KUKA KRL program: MyProgram_276().src

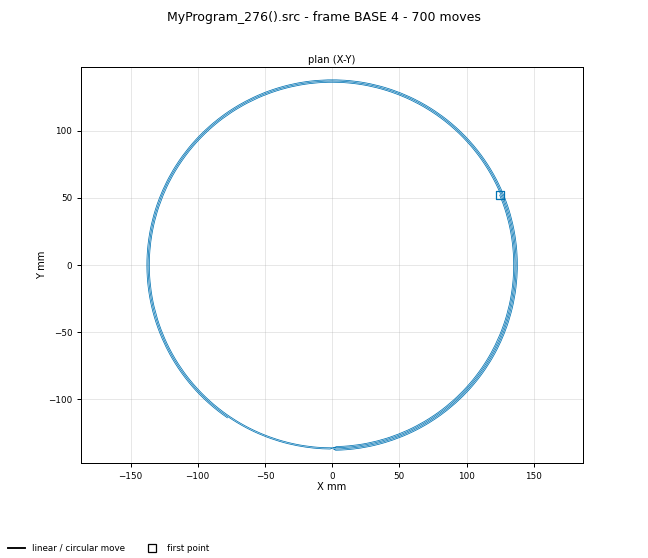
[picture p0: tool path of MyProgram_276().src in frame BASE 4, 700 of 700 moves have a stored position in this frame; points joined in program order, loops and branches not executed]
&ACCESS RVP
&REL 1
&PARAM TEMPLATE = C:\KRC\Roboter\Template\vorgabe
&PARAM EDITMASK = *
DEF MyProgram_276()
; ---- Setting reference (Base) ----
$BASE = BASE_DATA[4]

; --------------------------
; ---- Setting tool (TCP) ----
$TOOL = TOOL_DATA[3]
; --------------------------

$VEL.CP = VEL_APROX_PRINT
Startdeposition()
$VEL.CP = VEL_PRINT
LIN {X 124.6585,Y 52.0418,Z 172,A 23.3932,B 9.0147,C 0.1678,E1 9.1642,E2 428.0364} C_DIS
LIN {X 126.9033,Y 46.3017,Z 172,A 20.6618,B 9.0145,C 0.1775,E1 9.167,E2 430.7839} C_DIS
LIN {X 128.4598,Y 41.7937,Z 172,A 18.3883,B 9.0143,C 0.1885,E1 9.169,E2 433.0895} C_DIS
LIN {X 129.5892,Y 38.1419,Z 172,A 17.2072,B 9.0143,C 0.1833,E1 9.1699,E2 434.2181} C_DIS
LIN {X 130.4857,Y 34.952,Z 172,A 15.8377,B 9.0143,C 0.1864,E1 9.1709,E2 435.5844} C_DIS
LIN {X 131.283,Y 31.8269,Z 172,A 14.4299,B 9.0143,C 0.1911,E1 9.1719,E2 436.9981} C_DIS
LIN {X 132.2099,Y 27.7366,Z 172,A 12.5989,B 9.0141,C 0.1973,E1 9.173,E2 438.8371} C_DIS
LIN {X 132.9604,Y 23.8686,Z 172,A 11.0272,B 9.0141,C 0.1999,E1 9.1738,E2 440.3978} C_DIS
LIN {X 133.6197,Y 19.8624,Z 172,A 9.3104,B 9.0139,C 0.2047,E1 9.1745,E2 442.1155} C_DIS
LIN {X 134.1296,Y 16.0446,Z 172,A 7.7833,B 9.0139,C 0.207,E1 9.175,E2 443.6309} C_DIS
LIN {X 134.4806,Y 12.774,Z 172,A 6.3976,B 9.0138,C 0.2108,E1 9.1754,E2 445.0167} C_DIS
LIN {X 134.792,Y 8.9282,Z 172,A 4.7366,B 9.0137,C 0.2161,E1 9.1758,E2 446.6822} C_DIS
LIN {X 134.9785,Y 5.3889,Z 172,A 3.3382,B 9.0137,C 0.2181,E1 9.1759,E2 448.069} C_DIS
LIN {X 135.0733,Y 1.8859,Z 172,A 1.7806,B 9.0135,C 0.224,E1 9.176,E2 449.6368} C_DIS
LIN {X 135.0599,Y -2.6913,Z 172,A -0.171,B 9.0133,C 0.2299,E1 9.176,E2 451.5915} C_DIS
LIN {X 134.9407,Y -6.2819,Z 172,A -1.706,B 9.0133,C 0.2346,E1 9.1758,E2 453.1294} C_DIS
LIN {X 134.6433,Y -10.9355,Z 172,A -3.549,B 9.0131,C 0.2373,E1 9.1754,E2 454.9576} C_DIS
LIN {X 134.2842,Y -14.6974,Z 172,A -5.0801,B 9.0131,C 0.2403,E1 9.175,E2 456.4814} C_DIS
LIN {X 133.7732,Y -18.7889,Z 172,A -6.829,B 9.0129,C 0.2454,E1 9.1744,E2 458.2321} C_DIS
LIN {X 133.2905,Y -21.9519,Z 172,A -8.1831,B 9.0129,C 0.2492,E1 9.1738,E2 459.5872} C_DIS
LIN {X 132.6394,Y -25.593,Z 172,A -9.7051,B 9.0127,C 0.2527,E1 9.173,E2 461.105} C_DIS
LIN {X 131.7712,Y -29.7425,Z 172,A -11.5004,B 9.0126,C 0.2578,E1 9.1719,E2 462.9017} C_DIS
LIN {X 129.8103,Y -37.3868,Z 172,A -14.71,B 9.0124,C 0.2642,E1 9.1697,E2 466.0978} C_DIS
LIN {X 128.774,Y -40.81,Z 172,A -16.2644,B 9.0122,C 0.2693,E1 9.1684,E2 467.6584} C_DIS
LIN {X 127.6577,Y -44.1773,Z 172,A -17.8758,B 9.012,C 0.2758,E1 9.1669,E2 469.2845} C_DIS
LIN {X 126.162,Y -48.2881,Z 172,A -19.6376,B 9.012,C 0.2789,E1 9.1652,E2 471.0368} C_DIS
LIN {X 124.6634,Y -52.03,Z 172,A -21.2516,B 9.0119,C 0.2814,E1 9.1635,E2 472.6407} C_DIS
LIN {X 121.2699,Y -59.5127,Z 172,A -24.7108,B 9.0116,C 0.2902,E1 9.1595,E2 476.1004} C_DIS
LIN {X 119.7579,Y -62.4999,Z 172,A -26.052,B 9.0116,C 0.2921,E1 9.1577,E2 477.4333} C_DIS
LIN {X 118.3801,Y -65.0764,Z 172,A -27.7133,B 9.0111,C 0.3047,E1 9.1555,E2 479.1482} C_DIS
LIN {X 116.3933,Y -68.5656,Z 172,A -29.0606,B 9.0112,C 0.3012,E1 9.1536,E2 480.4534} C_DIS
LIN {X 114.0077,Y -72.464,Z 172,A -30.9991,B 9.0111,C 0.3061,E1 9.1507,E2 482.3939} C_DIS
LIN {X 111.4714,Y -76.3071,Z 172,A -33.1865,B 9.0107,C 0.316,E1 9.1473,E2 484.6123} C_DIS
LIN {X 109.2675,Y -79.4308,Z 172,A -34.4528,B 9.0109,C 0.3122,E1 9.1453,E2 485.8363} C_DIS
LIN {X 106.2421,Y -83.4339,Z 172,A -36.5817,B 9.0107,C 0.3172,E1 9.1416,E2 487.9674} C_DIS
LIN {X 103.9758,Y -86.2419,Z 172,A -38.2708,B 9.0104,C 0.3242,E1 9.1386,E2 489.6778} C_DIS
LIN {X 100.58,Y -90.1791,Z 172,A -40.272,B 9.0104,C 0.3247,E1 9.135,E2 491.6559} C_DIS
LIN {X 97.4489,Y -93.5543,Z 172,A -42.2111,B 9.0103,C 0.3287,E1 9.1312,E2 493.5953} C_DIS
LIN {X 93.0919,Y -97.8909,Z 172,A -44.7234,B 9.0102,C 0.3322,E1 9.1263,E2 496.0983} C_DIS
LIN {X 90.1601,Y -100.5971,Z 172,A -46.4322,B 9.01,C 0.336,E1 9.1227,E2 497.8109} C_DIS
LIN {X 86.9097,Y -103.4182,Z 172,A -48.2702,B 9.0099,C 0.3398,E1 9.1188,E2 499.6522} C_DIS
LIN {X 84.6977,Y -105.2375,Z 172,A -49.7894,B 9.0095,C 0.3487,E1 9.1154,E2 501.2104} C_DIS
LIN {X 81.5581,Y -107.6891,Z 172,A -51.1496,B 9.0097,C 0.3448,E1 9.1125,E2 502.5314} C_DIS
LIN {X 78.6638,Y -109.8209,Z 172,A -52.854,B 9.0094,C 0.3514,E1 9.1086,E2 504.2596} C_DIS
LIN {X 75.9077,Y -111.7438,Z 172,A -54.057,B 9.0095,C 0.3491,E1 9.1059,E2 505.4362} C_DIS
LIN {X 72.1688,Y -114.1941,Z 172,A -55.9191,B 9.0095,C 0.3515,E1 9.1015,E2 507.2958} C_DIS
LIN {X 68.5551,Y -116.3995,Z 172,A -57.8014,B 9.0093,C 0.3562,E1 9.097,E2 509.1904} C_DIS
LIN {X 62.8163,Y -119.5917,Z 172,A -60.4294,B 9.0093,C 0.3571,E1 9.0906,E2 511.8013} C_DIS
LIN {X 59.3078,Y -121.371,Z 172,A -62.0161,B 9.0092,C 0.3577,E1 9.0866,E2 513.3791} C_DIS
LIN {X 55.8404,Y -123.0061,Z 172,A -63.774,B 9.009,C 0.3626,E1 9.0821,E2 515.1549} C_DIS
LIN {X 52.2953,Y -124.5526,Z 172,A -65.2573,B 9.009,C 0.3614,E1 9.0783,E2 516.6198} C_DIS
LIN {X 49.4772,Y -125.6997,Z 172,A -66.9818,B 9.0086,C 0.3719,E1 9.0737,E2 518.3994} C_DIS
LIN {X 45.8436,Y -127.0688,Z 172,A -68.0618,B 9.009,C 0.362,E1 9.0711,E2 519.41} C_DIS
LIN {X 42.9727,Y -128.0685,Z 172,A -69.2939,B 9.009,C 0.3622,E1 9.0678,E2 520.636} C_DIS
LIN {X 39.7873,Y -129.0936,Z 172,A -70.8843,B 9.0088,C 0.3672,E1 9.0635,E2 522.2488} C_DIS
LIN {X 36.4926,Y -130.0632,Z 172,A -72.3381,B 9.0088,C 0.3684,E1 9.0596,E2 523.7033} C_DIS
LIN {X 33.6645,Y -130.8244,Z 172,A -73.6344,B 9.0087,C 0.3706,E1 9.0561,E2 525.0072} C_DIS
LIN {X 30.1406,Y -131.6803,Z 172,A -75.0314,B 9.0087,C 0.3689,E1 9.0524,E2 526.3877} C_DIS
LIN {X 27.0627,Y -132.3472,Z 172,A -76.4577,B 9.0087,C 0.3717,E1 9.0484,E2 527.8261} C_DIS
LIN {X 23.3507,Y -133.0531,Z 172,A -78.118,B 9.0085,C 0.3739,E1 9.0439,E2 529.4946} C_DIS
LIN {X 19.4834,Y -133.6739,Z 172,A -79.6978,B 9.0085,C 0.3732,E1 9.0395,E2 531.0654} C_DIS
LIN {X 15.8808,Y -134.1492,Z 172,A -81.1663,B 9.0085,C 0.3725,E1 9.0355,E2 532.5256} C_DIS
LIN {X 12.7336,Y -134.4845,Z 172,A -82.7735,B 9.0084,C 0.3783,E1 9.0309,E2 534.1666} C_DIS
LIN {X 8.3571,Y -134.8272,Z 172,A -85.0382,B 9.008,C 0.3868,E1 9.0245,E2 536.4822} C_DIS
LIN {X 3.3571,Y -135.0449,Z 172,A -86.6057,B 9.0084,C 0.3764,E1 9.0203,E2 537.9819} C_DIS
LIN {X 3.3571,Y -135.0449,Z 172,A -86.6057,B 9.0084,C 0.3764,E1 9.0203,E2 537.9819} C_DIS
Enddeposition()
LIN {X 0.9803,Y -135.9916,Z 172,A -87.1338,B 8.9369,C 0.374,E1 8.9473,E2 538.5052} C_DIS
Startdeposition()
$VEL.CP = VEL_PRINT
LIN {X 8.3933,Y -135.7358,Z 172,A -83.7774,B 8.9372,C 0.3688,E1 8.9567,E2 535.1182} C_DIS
LIN {X 14.9669,Y -135.1696,Z 172,A -80.9958,B 8.9372,C 0.3677,E1 8.9645,E2 532.3349} C_DIS
LIN {X 18.4168,Y -134.7443,Z 172,A -79.5305,B 8.9372,C 0.3669,E1 8.9685,E2 530.8687} C_DIS
LIN {X 23.3174,Y -133.9826,Z 172,A -77.4575,B 8.9372,C 0.366,E1 8.9742,E2 528.7965} C_DIS
LIN {X 26.1105,Y -133.4661,Z 172,A -76.2877,B 8.9372,C 0.3658,E1 8.9774,E2 527.6294} C_DIS
LIN {X 28.7703,Y -132.9168,Z 172,A -75.0894,B 8.9374,C 0.3638,E1 8.9807,E2 526.4234} C_DIS
LIN {X 32.1291,Y -132.1453,Z 172,A -73.607,B 8.9374,C 0.3621,E1 8.9848,E2 524.9361} C_DIS
LIN {X 36.5045,Y -131.0039,Z 172,A -71.6576,B 8.9375,C 0.3595,E1 8.9901,E2 522.9798} C_DIS
LIN {X 40.7735,Y -129.7401,Z 172,A -69.7219,B 8.9377,C 0.3564,E1 8.9952,E2 521.035} C_DIS
LIN {X 45.3449,Y -128.2148,Z 172,A -67.8777,B 8.9376,C 0.3582,E1 9.0001,E2 519.2131} C_DIS
LIN {X 47.9967,Y -127.2437,Z 172,A -66.6253,B 8.9376,C 0.3555,E1 9.0034,E2 517.9518} C_DIS
LIN {X 52.5626,Y -125.4262,Z 172,A -64.5866,B 8.9378,C 0.3537,E1 9.0086,E2 515.9154} C_DIS
LIN {X 55.8377,Y -124.0032,Z 172,A -63.0884,B 8.9378,C 0.3519,E1 9.0125,E2 514.4169} C_DIS
LIN {X 59.008,Y -122.5266,Z 172,A -61.6822,B 8.9378,C 0.3513,E1 9.016,E2 513.018} C_DIS
LIN {X 62.3605,Y -120.8563,Z 172,A -60.1169,B 8.9379,C 0.3494,E1 9.0199,E2 511.453} C_DIS
LIN {X 68.42,Y -117.5323,Z 172,A -57.3371,B 8.9379,C 0.3478,E1 9.0266,E2 508.6876} C_DIS
LIN {X 71.2892,Y -115.8143,Z 172,A -55.904,B 8.9381,C 0.345,E1 9.0301,E2 507.2502} C_DIS
LIN {X 74.2509,Y -113.9383,Z 172,A -54.2632,B 8.9383,C 0.3391,E1 9.034,E2 505.5873} C_DIS
LIN {X 77.8771,Y -111.4912,Z 172,A -52.6567,B 8.9383,C 0.341,E1 9.0376,E2 504.0091} C_DIS
LIN {X 80.2512,Y -109.7949,Z 172,A -51.2654,B 8.9385,C 0.3353,E1 9.0408,E2 502.5961} C_DIS
LIN {X 83.3437,Y -107.4658,Z 172,A -49.4889,B 8.9387,C 0.3291,E1 9.0448,E2 500.7995} C_DIS
LIN {X 87.2765,Y -104.2973,Z 172,A -47.4827,B 8.9387,C 0.3276,E1 9.0491,E2 498.8067} C_DIS
LIN {X 90.5204,Y -101.4948,Z 172,A -45.7122,B 8.9389,C 0.3248,E1 9.0528,E2 497.039} C_DIS
LIN {X 93.5734,Y -98.6874,Z 172,A -44.0017,B 8.9389,C 0.322,E1 9.0563,E2 495.3315} C_DIS
LIN {X 96.6359,Y -95.6902,Z 172,A -42.1996,B 8.9391,C 0.3182,E1 9.0598,E2 493.5281} C_DIS
LIN {X 99.6149,Y -92.5848,Z 172,A -40.4739,B 8.9391,C 0.3162,E1 9.0631,E2 491.8117} C_DIS
LIN {X 102.3677,Y -89.5319,Z 172,A -38.7632,B 8.9393,C 0.3128,E1 9.0663,E2 490.1019} C_DIS
LIN {X 105.0543,Y -86.3645,Z 172,A -36.9621,B 8.9395,C 0.3076,E1 9.0695,E2 488.2925} C_DIS
LIN {X 108.0127,Y -82.6337,Z 172,A -34.9947,B 8.9395,C 0.3037,E1 9.0729,E2 486.3279} C_DIS
LIN {X 110.4475,Y -79.3506,Z 172,A -33.1871,B 8.9398,C 0.2977,E1 9.0759,E2 484.5076} C_DIS
LIN {X 113.3117,Y -75.2041,Z 172,A -31.1844,B 8.9398,C 0.2952,E1 9.079,E2 482.5181} C_DIS
LIN {X 115.671,Y -71.5223,Z 172,A -29.3642,B 8.94,C 0.291,E1 9.0817,E2 480.6988} C_DIS
LIN {X 118.0971,Y -67.4399,Z 172,A -27.6092,B 8.94,C 0.2914,E1 9.0842,E2 478.9729} C_DIS
LIN {X 119.805,Y -64.3571,Z 172,A -25.9941,B 8.9402,C 0.2846,E1 9.0863,E2 477.3397} C_DIS
LIN {X 121.3273,Y -61.4352,Z 172,A -24.5834,B 8.9403,C 0.2805,E1 9.0881,E2 475.9247} C_DIS
LIN {X 123.3592,Y -57.2456,Z 172,A -22.5309,B 8.9406,C 0.2732,E1 9.0906,E2 473.8585} C_DIS
LIN {X 125.0219,Y -53.5193,Z 172,A -21.0781,B 8.9406,C 0.2746,E1 9.0922,E2 472.4377} C_DIS
LIN {X 126.3088,Y -50.407,Z 172,A -19.6713,B 8.9406,C 0.271,E1 9.0937,E2 471.031} C_DIS
LIN {X 127.472,Y -47.3873,Z 172,A -18.2657,B 8.9408,C 0.2663,E1 9.0951,E2 469.6186} C_DIS
LIN {X 128.6441,Y -44.1076,Z 172,A -16.8916,B 8.9408,C 0.2643,E1 9.0963,E2 468.2548} C_DIS
LIN {X 129.8056,Y -40.5673,Z 172,A -15.1381,B 8.9411,C 0.2558,E1 9.0978,E2 466.4765} C_DIS
LIN {X 131.1179,Y -36.0968,Z 172,A -13.1257,B 8.9413,C 0.2491,E1 9.0994,E2 464.4558} C_DIS
LIN {X 132.4689,Y -30.7709,Z 172,A -11.0904,B 8.9413,C 0.2489,E1 9.1007,E2 462.4535} C_DIS
LIN {X 133.2721,Y -27.0768,Z 172,A -9.5302,B 8.9413,C 0.2451,E1 9.1016,E2 460.8957} C_DIS
LIN {X 133.8593,Y -24.0065,Z 172,A -8.236,B 8.9415,C 0.2418,E1 9.1022,E2 459.6032} C_DIS
LIN {X 134.4917,Y -20.175,Z 172,A -6.6832,B 8.9415,C 0.239,E1 9.1029,E2 458.0593} C_DIS
LIN {X 134.8632,Y -17.5091,Z 172,A -5.5373,B 8.9416,C 0.2354,E1 9.1033,E2 456.9107} C_DIS
LIN {X 135.2914,Y -13.835,Z 172,A -4.0248,B 8.9417,C 0.232,E1 9.1038,E2 455.4025} C_DIS
LIN {X 135.5426,Y -11.0904,Z 172,A -2.8958,B 8.9417,C 0.2293,E1 9.1041,E2 454.2764} C_DIS
LIN {X 135.7847,Y -7.5962,Z 172,A -1.3594,B 8.9419,C 0.2237,E1 9.1043,E2 452.7309} C_DIS
LIN {X 135.9355,Y -4.0366,Z 172,A 0.0461,B 8.9419,C 0.2214,E1 9.1045,E2 451.336} C_DIS
LIN {X 135.9963,Y -0.4523,Z 172,A 1.6337,B 8.9421,C 0.2153,E1 9.1045,E2 449.7373} C_DIS
LIN {X 135.9434,Y 3.7502,Z 172,A 3.3637,B 8.9422,C 0.2111,E1 9.1045,E2 448.0107} C_DIS
LIN {X 135.7483,Y 8.1911,Z 172,A 5.1581,B 8.9423,C 0.2074,E1 9.1042,E2 446.2244} C_DIS
LIN {X 135.4785,Y 11.8487,Z 172,A 6.6754,B 8.9424,C 0.2036,E1 9.1038,E2 444.7093} C_DIS
LIN {X 135.0544,Y 15.9677,Z 172,A 8.4685,B 8.9425,C 0.1975,E1 9.1033,E2 442.9086} C_DIS
LIN {X 134.4792,Y 20.2557,Z 172,A 10.3046,B 8.9427,C 0.192,E1 9.1025,E2 441.0692} C_DIS
LIN {X 133.8343,Y 24.1459,Z 172,A 11.8398,B 8.9427,C 0.1901,E1 9.1018,E2 439.5484} C_DIS
LIN {X 133.0508,Y 28.1495,Z 172,A 13.5927,B 8.9428,C 0.1844,E1 9.1008,E2 437.7899} C_DIS
LIN {X 132.1905,Y 31.9415,Z 172,A 15.1026,B 8.9428,C 0.1827,E1 9.0999,E2 436.2947} C_DIS
LIN {X 131.3184,Y 35.3577,Z 172,A 16.5604,B 8.9429,C 0.1792,E1 9.0988,E2 434.8392} C_DIS
LIN {X 130.3402,Y 38.8125,Z 172,A 18.0645,B 8.943,C 0.1752,E1 9.0977,E2 433.3351} C_DIS
LIN {X 129.4646,Y 41.6361,Z 172,A 19.3291,B 8.943,C 0.1713,E1 9.0966,E2 432.0671} C_DIS
LIN {X 128.0477,Y 45.8088,Z 172,A 21.3563,B 8.9432,C 0.1624,E1 9.0947,E2 430.0172} C_DIS
LIN {X 126.1269,Y 50.858,Z 172,A 23.4459,B 8.9432,C 0.1605,E1 9.0926,E2 427.9494} C_DIS
LIN {X 124.8028,Y 54.0259,Z 172,A 24.8276,B 8.9433,C 0.1581,E1 9.0911,E2 426.5747} C_DIS
LIN {X 123.2607,Y 57.4588,Z 172,A 26.3457,B 8.9433,C 0.1554,E1 9.0893,E2 425.0641} C_DIS
LIN {X 121.8552,Y 60.3811,Z 172,A 27.7381,B 8.9434,C 0.1513,E1 9.0876,E2 423.6675} C_DIS
LIN {X 119.8353,Y 64.3008,Z 172,A 30.1722,B 8.9437,C 0.1338,E1 9.0843,E2 421.1603} C_DIS
LIN {X 117.2926,Y 68.8296,Z 172,A 31.7747,B 8.9437,C 0.1414,E1 9.0822,E2 419.6298} C_DIS
LIN {X 115.4746,Y 71.838,Z 172,A 33.2172,B 8.9437,C 0.1386,E1 9.0801,E2 418.1913} C_DIS
LIN {X 113.1263,Y 75.4818,Z 172,A 35.026,B 8.9437,C 0.1346,E1 9.0773,E2 416.3837} C_DIS
LIN {X 111.0831,Y 78.4578,Z 172,A 36.5285,B 8.9437,C 0.1314,E1 9.0749,E2 414.8827} C_DIS
LIN {X 108.5061,Y 81.9848,Z 172,A 38.3167,B 8.9437,C 0.1283,E1 9.0719,E2 413.1001} C_DIS
LIN {X 105.5397,Y 85.7704,Z 172,A 40.2983,B 8.9438,C 0.1247,E1 9.0685,E2 411.1232} C_DIS
LIN {X 102.9841,Y 88.822,Z 172,A 41.9694,B 8.9438,C 0.1212,E1 9.0655,E2 409.452} C_DIS
LIN {X 100.1879,Y 91.9645,Z 172,A 43.7162,B 8.9439,C 0.1179,E1 9.0622,E2 407.7077} C_DIS
LIN {X 97.4305,Y 94.8816,Z 172,A 45.3861,B 8.9439,C 0.1149,E1 9.059,E2 406.0399} C_DIS
LIN {X 94.4649,Y 97.8339,Z 172,A 47.1937,B 8.944,C 0.1104,E1 9.0554,E2 404.2262} C_DIS
LIN {X 91.2863,Y 100.8062,Z 172,A 49.031,B 8.944,C 0.1068,E1 9.0516,E2 402.3879} C_DIS
LIN {X 87.7545,Y 103.8961,Z 172,A 50.9507,B 8.9441,C 0.1043,E1 9.0475,E2 400.4748} C_DIS
LIN {X 84.3711,Y 106.6619,Z 172,A 52.7422,B 8.9441,C 0.1021,E1 9.0437,E2 398.6891} C_DIS
LIN {X 80.926,Y 109.2986,Z 172,A 54.5864,B 8.9441,C 0.0986,E1 9.0395,E2 396.8424} C_DIS
LIN {X 77.583,Y 111.6958,Z 172,A 56.3816,B 8.9442,C 0.0944,E1 9.0354,E2 395.0393} C_DIS
LIN {X 73.5369,Y 114.4005,Z 172,A 58.3537,B 8.9442,C 0.0928,E1 9.0308,E2 393.0766} C_DIS
LIN {X 68.4098,Y 117.5384,Z 172,A 60.8845,B 8.9442,C 0.0892,E1 9.0248,E2 390.5459} C_DIS
LIN {X 64.5562,Y 119.698,Z 172,A 62.7253,B 8.9442,C 0.087,E1 9.0203,E2 388.7074} C_DIS
LIN {X 61.1621,Y 121.4664,Z 172,A 64.1782,B 8.9442,C 0.0882,E1 9.0167,E2 387.274} C_DIS
LIN {X 58.6285,Y 122.7079,Z 172,A 65.4068,B 8.9442,C 0.0859,E1 9.0136,E2 386.0406} C_DIS
LIN {X 55.1332,Y 124.3184,Z 172,A 67.1072,B 8.9443,C 0.0824,E1 9.0093,E2 384.3306} C_DIS
LIN {X 49.8291,Y 126.5384,Z 172,A 69.3004,B 8.9443,C 0.0845,E1 9.0037,E2 382.1657} C_DIS
LIN {X 46.8574,Y 127.6697,Z 172,A 70.7008,B 8.9443,C 0.0819,E1 9,E2 380.758} C_DIS
LIN {X 44.2389,Y 128.5985,Z 172,A 71.8884,B 8.9443,C 0.0805,E1 8.9968,E2 379.5685} C_DIS
LIN {X 40.7163,Y 129.7584,Z 172,A 73.7115,B 8.9444,C 0.0739,E1 8.9919,E2 377.7136} C_DIS
LIN {X 36.7718,Y 130.9291,Z 172,A 75.1533,B 8.9444,C 0.0784,E1 8.9881,E2 376.3079} C_DIS
LIN {X 33.2363,Y 131.8711,Z 172,A 76.7,B 8.9444,C 0.0772,E1 8.9839,E2 374.7609} C_DIS
LIN {X 29.7396,Y 132.7044,Z 172,A 78.1979,B 8.9444,C 0.0766,E1 8.9799,E2 373.2654} C_DIS
LIN {X 26.9398,Y 133.3,Z 172,A 79.4044,B 8.9444,C 0.0759,E1 8.9766,E2 372.0591} C_DIS
LIN {X 23.4766,Y 133.9541,Z 172,A 80.8802,B 8.9444,C 0.0753,E1 8.9725,E2 370.5848} C_DIS
LIN {X 19.7835,Y 134.5494,Z 172,A 82.5293,B 8.9444,C 0.0732,E1 8.968,E2 368.9273} C_DIS
LIN {X 16.0797,Y 135.041,Z 172,A 84.068,B 8.9444,C 0.0734,E1 8.9637,E2 367.3935} C_DIS
LIN {X 12.6788,Y 135.4031,Z 172,A 85.4668,B 8.9444,C 0.0738,E1 8.9598,E2 366.0003} C_DIS
LIN {X 8.8031,Y 135.7106,Z 172,A 87.1984,B 8.9444,C 0.0717,E1 8.955,E2 364.2579} C_DIS
LIN {X 4.8357,Y 135.9099,Z 172,A 88.9036,B 8.9444,C 0.0709,E1 8.9502,E2 362.5495} C_DIS
LIN {X 0.1298,Y 135.9965,Z 172,A 90.7352,B 8.9444,C 0.0738,E1 8.9451,E2 360.7374} C_DIS
LIN {X -3.1315,Y 135.9606,Z 172,A 92.2682,B 8.9444,C 0.0709,E1 8.9408,E2 359.1856} C_DIS
LIN {X -6.9147,Y 135.8192,Z 172,A 93.8022,B 8.9444,C 0.0723,E1 8.9366,E2 357.6598} C_DIS
LIN {X -10.4014,Y 135.5977,Z 172,A 95.172,B 8.9444,C 0.0745,E1 8.9328,E2 356.3033} C_DIS
LIN {X -13.7839,Y 135.2969,Z 172,A 96.6221,B 8.9444,C 0.0746,E1 8.9287,E2 354.8517} C_DIS
LIN {X -16.2942,Y 135.0154,Z 172,A 97.7336,B 8.9444,C 0.0741,E1 8.9256,E2 353.7349} C_DIS
LIN {X -20.1414,Y 134.4969,Z 172,A 99.4664,B 8.9444,C 0.073,E1 8.9208,E2 351.9912} C_DIS
LIN {X -23.9244,Y 133.874,Z 172,A 100.9521,B 8.9444,C 0.0762,E1 8.9168,E2 350.5222} C_DIS
LIN {X -27.7712,Y 133.1308,Z 172,A 102.6062,B 8.9444,C 0.0771,E1 8.9123,E2 348.8688} C_DIS
LIN {X -30.4539,Y 132.5413,Z 172,A 103.8168,B 8.9444,C 0.0769,E1 8.9089,E2 347.6523} C_DIS
LIN {X -34.1332,Y 131.6435,Z 172,A 105.6608,B 8.9444,C 0.0736,E1 8.9039,E2 345.7792} C_DIS
LIN {X -38.1097,Y 130.5459,Z 172,A 107.1853,B 8.9444,C 0.0789,E1 8.8999,E2 344.2819} C_DIS
LIN {X -41.5973,Y 129.4769,Z 172,A 108.6844,B 8.9444,C 0.0809,E1 8.8959,E2 342.7885} C_DIS
LIN {X -45.1968,Y 128.2664,Z 172,A 110.2632,B 8.9444,C 0.0828,E1 8.8917,E2 341.2135} C_DIS
LIN {X -49.4907,Y 126.6699,Z 172,A 112.0002,B 8.9443,C 0.0883,E1 8.8872,E2 339.5013} C_DIS
LIN {X -51.7786,Y 125.7536,Z 172,A 113.2216,B 8.9443,C 0.0862,E1 8.884,E2 338.2587} C_DIS
LIN {X -55.1158,Y 124.3261,Z 172,A 114.8798,B 8.9443,C 0.0857,E1 8.8797,E2 336.5859} C_DIS
LIN {X -62.7864,Y 120.6343,Z 172,A 118.304,B 8.9443,C 0.0933,E1 8.8712,E2 333.1846} C_DIS
LIN {X -65.4799,Y 119.1957,Z 172,A 120.1297,B 8.9443,C 0.0856,E1 8.8666,E2 331.2942} C_DIS
LIN {X -68.7371,Y 117.347,Z 172,A 121.1751,B 8.9442,C 0.0973,E1 8.8642,E2 330.3151} C_DIS
LIN {X -71.2105,Y 115.8627,Z 172,A 122.6152,B 8.9442,C 0.0952,E1 8.8607,E2 328.8488} C_DIS
LIN {X -74.8418,Y 113.5508,Z 172,A 124.4386,B 8.9442,C 0.098,E1 8.8564,E2 327.0258} C_DIS
LIN {X -81.3118,Y 109.0113,Z 172,A 127.7077,B 8.9442,C 0.1047,E1 8.849,E2 323.7673} C_DIS
LIN {X -83.6312,Y 107.2429,Z 172,A 129.084,B 8.9442,C 0.1044,E1 8.8459,E2 322.3742} C_DIS
LIN {X -86.8394,Y 104.6613,Z 172,A 130.7986,B 8.9441,C 0.108,E1 8.8422,E2 320.6637} C_DIS
LIN {X -91.136,Y 100.9427,Z 172,A 133.2526,B 8.9441,C 0.1116,E1 8.8371,E2 318.2047} C_DIS
LIN {X -94.6707,Y 97.6347,Z 172,A 135.3219,B 8.944,C 0.1152,E1 8.8329,E2 316.1337} C_DIS
LIN {X -97.9379,Y 94.3575,Z 172,A 137.7627,B 8.944,C 0.111,E1 8.828,E2 313.6345} C_DIS
LIN {X -101.1098,Y 90.9503,Z 172,A 138.9738,B 8.9438,C 0.1279,E1 8.8259,E2 312.5172} C_DIS
LIN {X -103.4317,Y 88.3008,Z 172,A 140.7247,B 8.9438,C 0.1267,E1 8.8227,E2 310.7353} C_DIS
LIN {X -106.1499,Y 85.0143,Z 172,A 142.6063,B 8.9438,C 0.1294,E1 8.8193,E2 308.8452} C_DIS
LIN {X -108.8218,Y 81.5664,Z 172,A 144.4835,B 8.9438,C 0.1331,E1 8.8162,E2 306.9651} C_DIS
LIN {X -111.6887,Y 77.5932,Z 172,A 146.5348,B 8.9436,C 0.1382,E1 8.8128,E2 304.9175} C_DIS
LIN {X -114.1445,Y 73.9333,Z 172,A 148.4574,B 8.9436,C 0.1417,E1 8.8099,E2 302.9887} C_DIS
LIN {X -116.6202,Y 69.9639,Z 172,A 150.4114,B 8.9436,C 0.1469,E1 8.807,E2 301.0388} C_DIS
LIN {X -118.6719,Y 66.4237,Z 172,A 152.406,B 8.9436,C 0.1469,E1 8.8043,E2 299.0128} C_DIS
LIN {X -121.3622,Y 61.3668,Z 172,A 154.5518,B 8.9433,C 0.1574,E1 8.8015,E2 296.9023} C_DIS
LIN {X -122.7459,Y 58.5488,Z 172,A 155.9178,B 8.9433,C 0.1602,E1 8.7999,E2 295.5323} C_DIS
LIN {X -124.4783,Y 54.7755,Z 172,A 157.6643,B 8.9433,C 0.1649,E1 8.7979,E2 293.7881} C_DIS
LIN {X -125.6097,Y 52.1232,Z 172,A 158.9637,B 8.9432,C 0.1668,E1 8.7965,E2 292.4795} C_DIS
LIN {X -128.9819,Y 43.1075,Z 172,A 163.0962,B 8.943,C 0.1767,E1 8.7925,E2 288.3418} C_DIS
LIN {X -130.1217,Y 39.5346,Z 172,A 164.6608,B 8.9429,C 0.1814,E1 8.7912,E2 286.7808} C_DIS
LIN {X -131.1093,Y 36.1274,Z 172,A 166.1526,B 8.9428,C 0.1856,E1 8.7901,E2 285.291} C_DIS
LIN {X -131.9308,Y 33.001,Z 172,A 167.4861,B 8.9428,C 0.1899,E1 8.7892,E2 283.9623} C_DIS
LIN {X -132.7225,Y 29.6605,Z 172,A 169.063,B 8.9427,C 0.1919,E1 8.7882,E2 282.3708} C_DIS
LIN {X -133.5936,Y 25.4434,Z 172,A 170.9015,B 8.9426,C 0.1967,E1 8.7872,E2 280.5311} C_DIS
LIN {X -134.2716,Y 21.5963,Z 172,A 172.4983,B 8.9424,C 0.2023,E1 8.7864,E2 278.942} C_DIS
LIN {X -134.8924,Y 17.2868,Z 172,A 174.3445,B 8.9424,C 0.2073,E1 8.7857,E2 277.0961} C_DIS
LIN {X -135.256,Y 14.1633,Z 172,A 175.6979,B 8.9422,C 0.2107,E1 8.7853,E2 275.7405} C_DIS
LIN {X -135.5549,Y 10.9443,Z 172,A 177.2445,B 8.9422,C 0.2117,E1 8.7849,E2 274.1725} C_DIS
LIN {X -135.8238,Y 6.8233,Z 172,A 178.8985,B 8.9421,C 0.2181,E1 8.7847,E2 272.5306} C_DIS
LIN {X -135.9554,Y 3.3185,Z 172,A -179.488,B 8.9421,C 0.2202,E1 8.7845,E2 270.9018} C_DIS
LIN {X -135.9949,Y -0.6567,Z 172,A -177.8433,B 8.9419,C 0.2256,E1 8.7845,E2 269.2624} C_DIS
LIN {X -135.9129,Y -4.7593,Z 172,A -176.1309,B 8.9418,C 0.2308,E1 8.7847,E2 267.5536} C_DIS
LIN {X -135.7388,Y -8.3457,Z 172,A -174.6014,B 8.9416,C 0.2349,E1 8.7849,E2 266.0234} C_DIS
LIN {X -135.4472,Y -12.219,Z 172,A -172.7588,B 8.9416,C 0.2363,E1 8.7853,E2 264.1568} C_DIS
LIN {X -134.9656,Y -16.7119,Z 172,A -171.069,B 8.9414,C 0.2452,E1 8.7859,E2 262.4951} C_DIS
LIN {X -134.5771,Y -19.5896,Z 172,A -169.7003,B 8.9414,C 0.2464,E1 8.7864,E2 261.1095} C_DIS
LIN {X -133.9182,Y -23.6774,Z 172,A -167.8931,B 8.9412,C 0.2503,E1 8.7872,E2 259.2958} C_DIS
LIN {X -133.1594,Y -27.6308,Z 172,A -166.306,B 8.941,C 0.2569,E1 8.7881,E2 257.7237} C_DIS
LIN {X -132.419,Y -30.9891,Z 172,A -164.5382,B 8.941,C 0.2558,E1 8.7892,E2 255.9174} C_DIS
LIN {X -129.8539,Y -40.4092,Z 172,A -160.6055,B 8.9407,C 0.2702,E1 8.7922,E2 252.0106} C_DIS
LIN {X -128.5074,Y -44.5017,Z 172,A -158.6716,B 8.9406,C 0.2731,E1 8.7939,E2 250.0632} C_DIS
LIN {X -127.214,Y -48.076,Z 172,A -157.1373,B 8.9404,C 0.2785,E1 8.7954,E2 248.5384} C_DIS
LIN {X -126.0077,Y -51.1538,Z 172,A -155.7306,B 8.9403,C 0.282,E1 8.7969,E2 247.1309} C_DIS
LIN {X -124.7203,Y -54.2168,Z 172,A -154.3198,B 8.9402,C 0.2855,E1 8.7984,E2 245.7197} C_DIS
LIN {X -122.9977,Y -58.0219,Z 172,A -152.3744,B 8.9402,C 0.287,E1 8.8007,E2 243.7524} C_DIS
LIN {X -121.2416,Y -61.6035,Z 172,A -150.7233,B 8.94,C 0.2918,E1 8.8028,E2 242.1059} C_DIS
LIN {X -119.0189,Y -65.7997,Z 172,A -148.7054,B 8.9398,C 0.2965,E1 8.8055,E2 240.0871} C_DIS
LIN {X -116.7492,Y -69.7476,Z 172,A -146.8001,B 8.9397,C 0.3014,E1 8.8082,E2 238.1846} C_DIS
LIN {X -114.4724,Y -73.4245,Z 172,A -144.5131,B 8.9397,C 0.2979,E1 8.8117,E2 235.8402} C_DIS
LIN {X -112.1292,Y -76.9553,Z 172,A -143.3544,B 8.9393,C 0.3128,E1 8.8134,E2 234.761} C_DIS
LIN {X -110.4158,Y -79.395,Z 172,A -141.6107,B 8.9395,C 0.3074,E1 8.8163,E2 232.9569} C_DIS
LIN {X -108.4822,Y -82.0164,Z 172,A -140.495,B 8.9392,C 0.3148,E1 8.8181,E2 231.8741} C_DIS
LIN {X -106.0275,Y -85.1663,Z 172,A -138.7806,B 8.9391,C 0.318,E1 8.8211,E2 230.1564} C_DIS
LIN {X -103.3516,Y -88.395,Z 172,A -136.8963,B 8.9391,C 0.3198,E1 8.8245,E2 228.258} C_DIS
LIN {X -100.3177,Y -91.8233,Z 172,A -134.9478,B 8.9389,C 0.3235,E1 8.8281,E2 226.3078} C_DIS
LIN {X -97.2912,Y -95.024,Z 172,A -133.0804,B 8.9388,C 0.327,E1 8.8318,E2 224.4396} C_DIS
LIN {X -94.269,Y -98.0234,Z 172,A -131.2509,B 8.9387,C 0.3299,E1 8.8354,E2 222.6062} C_DIS
LIN {X -91.1999,Y -100.8846,Z 172,A -129.5387,B 8.9385,C 0.3342,E1 8.8389,E2 220.9015} C_DIS
LIN {X -88.0111,Y -103.678,Z 172,A -127.6328,B 8.9385,C 0.3353,E1 8.843,E2 218.9809} C_DIS
LIN {X -84.6326,Y -106.4537,Z 172,A -125.8682,B 8.9383,C 0.3399,E1 8.8468,E2 217.2264} C_DIS
LIN {X -81.07,Y -109.1914,Z 172,A -123.7344,B 8.9383,C 0.3387,E1 8.8516,E2 215.0626} C_DIS
LIN {X -78.4658,Y -111.0774,Z 172,A -122.7462,B 8.938,C 0.3474,E1 8.8538,E2 214.1209} C_DIS
LIN {X -75.6552,Y -113.0106,Z 172,A -121.0998,B 8.938,C 0.3459,E1 8.8577,E2 212.4483} C_DIS
LIN {X -71.243,Y -115.8427,Z 172,A -119.128,B 8.9378,C 0.3534,E1 8.8622,E2 210.5067} C_DIS
LIN {X -68.4324,Y -117.5253,Z 172,A -117.5337,B 8.9378,C 0.3514,E1 8.8661,E2 208.8855} C_DIS
LIN {X -64.8066,Y -119.563,Z 172,A -115.696,B 8.9378,C 0.3521,E1 8.8707,E2 207.037} C_DIS
LIN {X -61.7544,Y -121.1649,Z 172,A -114.2671,B 8.9378,C 0.3543,E1 8.8742,E2 205.6111} C_DIS
LIN {X -57.9093,Y -123.0515,Z 172,A -112.3867,B 8.9378,C 0.355,E1 8.879,E2 203.721} C_DIS
LIN {X -52.9501,Y -125.2644,Z 172,A -110.3392,B 8.9374,C 0.3618,E1 8.8841,E2 201.7038} C_DIS
LIN {X -49.0272,Y -126.8501,Z 172,A -108.451,B 8.9374,C 0.3616,E1 8.8891,E2 199.8021} C_DIS
LIN {X -45.8817,Y -128.0214,Z 172,A -106.981,B 8.9374,C 0.3618,E1 8.8929,E2 198.3248} C_DIS
LIN {X -40.7787,Y -129.7384,Z 172,A -104.7754,B 8.9374,C 0.3648,E1 8.8988,E2 196.127} C_DIS
LIN {X -37.3954,Y -130.7547,Z 172,A -103.2734,B 8.9373,C 0.3656,E1 8.9028,E2 194.6229} C_DIS
LIN {X -32.6529,Y -132.0191,Z 172,A -101.1938,B 8.9373,C 0.3666,E1 8.9084,E2 192.5414} C_DIS
LIN {X -28.561,Y -132.962,Z 172,A -99.3661,B 8.9373,C 0.3664,E1 8.9134,E2 190.7058} C_DIS
LIN {X -24.4355,Y -133.7825,Z 172,A -97.5201,B 8.9373,C 0.3657,E1 8.9185,E2 188.8498} C_DIS
LIN {X -20.5102,Y -134.4398,Z 172,A -95.922,B 8.9373,C 0.3678,E1 8.9229,E2 187.2612} C_DIS
LIN {X -14.3847,Y -135.2322,Z 172,A -93.3621,B 8.9371,C 0.3693,E1 8.93,E2 184.7059} C_DIS
LIN {X -11.2036,Y -135.533,Z 172,A -91.3674,B 8.9377,C 0.3567,E1 8.9358,E2 182.6278} C_DIS
LIN {X -6.0611,Y -135.8621,Z 172,A -89.8547,B 8.9371,C 0.3697,E1 8.9398,E2 181.1984} C_DIS
LIN {X 0.9803,Y -135.9916,Z 172,A -87.1317,B 8.9369,C 0.3744,E1 8.9473,E2 178.5052} C_DIS
Enddeposition()
LIN {X 0.9803,Y -135.9916,Z 172,A -87.1317,B 8.9369,C 0.3744,E1 8.9473,E2 178.5052} C_DIS
Startdeposition()
$VEL.CP = VEL_PRINT
LIN {X -1.516,Y -136.898,Z 172,A -88.4457,B 8.8637,C 0.3865,E1 8.8707,E2 179.9091} C_DIS
LIN {X -4.5679,Y -136.8302,Z 172,A -89.7257,B 8.8637,C 0.3866,E1 8.8672,E2 181.19} C_DIS
LIN {X -7.345,Y -136.7079,Z 172,A -90.892,B 8.8637,C 0.3866,E1 8.8639,E2 182.3571} C_DIS
LIN {X -10.4422,Y -136.5062,Z 172,A -92.194,B 8.8637,C 0.3866,E1 8.8603,E2 183.66} C_DIS
LIN {X -13.8641,Y -136.2026,Z 172,A -93.6355,B 8.8637,C 0.3865,E1 8.8563,E2 185.1026} C_DIS
LIN {X -17.0023,Y -135.8466,Z 172,A -94.9611,B 8.8637,C 0.3863,E1 8.8526,E2 186.4291} C_DIS
LIN {X -19.6184,Y -135.4914,Z 172,A -96.1215,B 8.8637,C 0.387,E1 8.8494,E2 187.5969} C_DIS
LIN {X -23.0157,Y -134.9565,Z 172,A -97.5197,B 8.8637,C 0.3857,E1 8.8455,E2 188.9903} C_DIS
LIN {X -26.2102,Y -134.3726,Z 172,A -98.8741,B 8.8638,C 0.3851,E1 8.8418,E2 190.3446} C_DIS
LIN {X -29.3786,Y -133.7156,Z 172,A -100.259,B 8.8638,C 0.385,E1 8.838,E2 191.7337} C_DIS
LIN {X -32.5697,Y -132.9743,Z 172,A -101.6171,B 8.8638,C 0.384,E1 8.8343,E2 193.0905} C_DIS
LIN {X -35.5272,Y -132.2141,Z 172,A -102.9288,B 8.8638,C 0.3838,E1 8.8308,E2 194.4067} C_DIS
LIN {X -39.2673,Y -131.1543,Z 172,A -104.537,B 8.8639,C 0.3824,E1 8.8264,E2 196.0129} C_DIS
LIN {X -42.457,Y -130.1567,Z 172,A -105.9433,B 8.8639,C 0.3814,E1 8.8227,E2 197.4204} C_DIS
LIN {X -45.3733,Y -129.1675,Z 172,A -107.2187,B 8.864,C 0.3801,E1 8.8193,E2 198.6942} C_DIS
LIN {X -48.4365,Y -128.0498,Z 172,A -108.6203,B 8.864,C 0.3796,E1 8.8157,E2 200.1007} C_DIS
LIN {X -51.9726,Y -126.6579,Z 172,A -110.2148,B 8.8641,C 0.3781,E1 8.8115,E2 201.696} C_DIS
LIN {X -54.8107,Y -125.454,Z 172,A -111.5145,B 8.8641,C 0.3769,E1 8.8082,E2 202.9969} C_DIS
LIN {X -57.819,Y -124.0957,Z 172,A -112.9184,B 8.8642,C 0.3758,E1 8.8046,E2 204.4036} C_DIS
LIN {X -61.039,Y -122.5444,Z 172,A -114.4136,B 8.8642,C 0.374,E1 8.8009,E2 205.8988} C_DIS
LIN {X -64.1157,Y -120.9631,Z 172,A -115.7002,B 8.8645,C 0.3694,E1 8.7977,E2 207.165} C_DIS
LIN {X -67.1135,Y -119.3271,Z 172,A -117.3719,B 8.8644,C 0.3719,E1 8.7936,E2 208.8673} C_DIS
LIN {X -70.8887,Y -117.1237,Z 172,A -119.193,B 8.8644,C 0.3692,E1 8.7892,E2 210.6872} C_DIS
LIN {X -74.0381,Y -115.1591,Z 172,A -120.717,B 8.8646,C 0.3664,E1 8.7856,E2 212.2074} C_DIS
LIN {X -77.2468,Y -113.0318,Z 172,A -122.4544,B 8.8646,C 0.3662,E1 8.7815,E2 213.9604} C_DIS
LIN {X -80.561,Y -110.694,Z 172,A -124.1318,B 8.8647,C 0.3631,E1 8.7777,E2 215.6351} C_DIS
LIN {X -84.0831,Y -108.043,Z 172,A -125.9945,B 8.8648,C 0.3603,E1 8.7736,E2 217.4997} C_DIS
LIN {X -87.5248,Y -105.2742,Z 172,A -127.8197,B 8.865,C 0.3567,E1 8.7697,E2 219.3214} C_DIS
LIN {X -90.6851,Y -102.5641,Z 172,A -129.6251,B 8.865,C 0.3546,E1 8.7658,E2 221.1343} C_DIS
LIN {X -93.7204,Y -99.7986,Z 172,A -131.4095,B 8.8652,C 0.3525,E1 8.7622,E2 222.9265} C_DIS
LIN {X -96.6853,Y -96.9289,Z 172,A -133.0608,B 8.8653,C 0.3478,E1 8.7589,E2 224.5678} C_DIS
LIN {X -99.399,Y -94.144,Z 172,A -134.7931,B 8.8653,C 0.3464,E1 8.7555,E2 226.3126} C_DIS
LIN {X -102.1627,Y -91.1375,Z 172,A -136.4854,B 8.8655,C 0.3425,E1 8.7524,E2 228.0023} C_DIS
LIN {X -105.0403,Y -87.8054,Z 172,A -138.3538,B 8.8657,C 0.339,E1 8.749,E2 229.873} C_DIS
LIN {X -107.8318,Y -84.3537,Z 172,A -140.1876,B 8.8658,C 0.3345,E1 8.7458,E2 231.703} C_DIS
LIN {X -110.334,Y -81.053,Z 172,A -142.0061,B 8.8659,C 0.332,E1 8.7427,E2 233.5314} C_DIS
LIN {X -113.0318,Y -77.2468,Z 172,A -143.9007,B 8.8661,C 0.3265,E1 8.7397,E2 235.4178} C_DIS
LIN {X -115.1591,Y -74.0381,Z 172,A -145.6245,B 8.8662,C 0.3246,E1 8.7371,E2 237.1548} C_DIS
LIN {X -117.4643,Y -70.3235,Z 172,A -147.4883,B 8.8663,C 0.3207,E1 8.7344,E2 239.0219} C_DIS
LIN {X -119.5595,Y -66.7,Z 172,A -149.207,B 8.8665,C 0.3158,E1 8.732,E2 240.7355} C_DIS
LIN {X -121.6118,Y -62.8804,Z 172,A -151.0035,B 8.8667,C 0.311,E1 8.7296,E2 242.5286} C_DIS
LIN {X -122.9405,Y -60.2363,Z 172,A -152.3008,B 8.8667,C 0.3087,E1 8.728,E2 243.8324} C_DIS
LIN {X -124.6223,Y -56.6803,Z 172,A -153.929,B 8.8669,C 0.3042,E1 8.7261,E2 245.4574} C_DIS
LIN {X -125.9851,Y -53.5822,Z 172,A -155.3602,B 8.867,C 0.3007,E1 8.7245,E2 246.8894} C_DIS
LIN {X -127.1703,Y -50.7014,Z 172,A -156.696,B 8.8671,C 0.2978,E1 8.7231,E2 248.2282} C_DIS
LIN {X -128.5026,Y -47.2278,Z 172,A -158.2682,B 8.8673,C 0.2939,E1 8.7216,E2 249.8013} C_DIS
LIN {X -129.5192,Y -44.3587,Z 172,A -159.5669,B 8.8673,C 0.2908,E1 8.7204,E2 251.1021} C_DIS
LIN {X -130.567,Y -41.1728,Z 172,A -160.9843,B 8.8675,C 0.2872,E1 8.7192,E2 252.5201} C_DIS
LIN {X -131.5308,Y -37.9813,Z 172,A -162.4204,B 8.8675,C 0.284,E1 8.718,E2 253.9603} C_DIS
LIN {X -132.4942,Y -34.4769,Z 172,A -163.9442,B 8.8677,C 0.2798,E1 8.7169,E2 255.4833} C_DIS
LIN {X -133.1754,Y -31.7353,Z 172,A -165.1336,B 8.8678,C 0.2766,E1 8.7161,E2 256.6726} C_DIS
LIN {X -133.9547,Y -28.2711,Z 172,A -166.6594,B 8.8679,C 0.2731,E1 8.7152,E2 258.2021} C_DIS
LIN {X -134.5617,Y -25.2211,Z 172,A -167.973,B 8.868,C 0.2696,E1 8.7145,E2 259.5161} C_DIS
LIN {X -135.1381,Y -21.9274,Z 172,A -169.3513,B 8.8682,C 0.2653,E1 8.7139,E2 260.8907} C_DIS
LIN {X -135.5478,Y -19.2239,Z 172,A -170.5949,B 8.8682,C 0.2636,E1 8.7134,E2 262.1455} C_DIS
LIN {X -135.9976,Y -15.7366,Z 172,A -172.0487,B 8.8683,C 0.2591,E1 8.7129,E2 263.5959} C_DIS
LIN {X -136.3235,Y -12.6054,Z 172,A -173.3916,B 8.8684,C 0.2557,E1 8.7125,E2 264.9407} C_DIS
LIN {X -136.5632,Y -9.6625,Z 172,A -174.634,B 8.8685,C 0.2522,E1 8.7123,E2 266.1829} C_DIS
LIN {X -136.7703,Y -6.1033,Z 172,A -176.1557,B 8.8687,C 0.2484,E1 8.712,E2 267.7069} C_DIS
LIN {X -136.8644,Y -3.3361,Z 172,A -177.35,B 8.8687,C 0.2456,E1 8.712,E2 268.9045} C_DIS
LIN {X -136.9051,Y 0.5094,Z 172,A -179.0786,B 8.8688,C 0.2429,E1 8.712,E2 270.6464} C_DIS
LIN {X -136.8481,Y 3.9233,Z 172,A 179.5302,B 8.8689,C 0.2381,E1 8.712,E2 272.0316} C_DIS
LIN {X -136.7079,Y 7.345,Z 172,A 178.1152,B 8.869,C 0.2337,E1 8.7122,E2 273.4429} C_DIS
LIN {X -136.5062,Y 10.4422,Z 172,A 176.7917,B 8.8691,C 0.2303,E1 8.7124,E2 274.7682} C_DIS
LIN {X -136.2026,Y 13.8641,Z 172,A 175.3269,B 8.8692,C 0.2266,E1 8.7128,E2 276.235} C_DIS
LIN {X -135.864,Y 16.8561,Z 172,A 174.0495,B 8.8693,C 0.2232,E1 8.7133,E2 277.5133} C_DIS
LIN {X -135.4145,Y 20.1565,Z 172,A 172.6236,B 8.8694,C 0.2197,E1 8.7138,E2 278.9417} C_DIS
LIN {X -134.9565,Y 23.0157,Z 172,A 171.369,B 8.8694,C 0.2169,E1 8.7144,E2 280.2004} C_DIS
LIN {X -134.3168,Y 26.5022,Z 172,A 169.8782,B 8.8696,C 0.2128,E1 8.7152,E2 281.6906} C_DIS
LIN {X -133.7672,Y 29.1394,Z 172,A 168.6745,B 8.8696,C 0.2108,E1 8.7159,E2 282.9025} C_DIS
LIN {X -132.9743,Y 32.5697,Z 172,A 167.2291,B 8.8697,C 0.2061,E1 8.7168,E2 284.343} C_DIS
LIN {X -132.1511,Y 35.7635,Z 172,A 165.824,B 8.8698,C 0.2026,E1 8.7178,E2 285.7497} C_DIS
LIN {X -131.1543,Y 39.2673,Z 172,A 164.2724,B 8.8698,C 0.1988,E1 8.719,E2 287.3032} C_DIS
LIN {X -130.1567,Y 42.457,Z 172,A 162.8494,B 8.87,C 0.1953,E1 8.7202,E2 288.7277} C_DIS
LIN {X -129.0751,Y 45.6399,Z 172,A 161.4179,B 8.87,C 0.1918,E1 8.7215,E2 290.1608} C_DIS
LIN {X -128.0243,Y 48.5046,Z 172,A 160.1181,B 8.8701,C 0.1887,E1 8.7228,E2 291.462} C_DIS
LIN {X -126.8852,Y 51.4086,Z 172,A 158.7835,B 8.8701,C 0.1856,E1 8.7242,E2 292.7987} C_DIS
LIN {X -125.454,Y 54.8107,Z 172,A 157.2196,B 8.8703,C 0.1818,E1 8.7259,E2 294.3635} C_DIS
LIN {X -124.0415,Y 57.9363,Z 172,A 155.7602,B 8.8703,C 0.1784,E1 8.7276,E2 295.8243} C_DIS
LIN {X -122.5444,Y 61.039,Z 172,A 154.2949,B 8.8703,C 0.175,E1 8.7294,E2 297.291} C_DIS
LIN {X -120.9631,Y 64.1157,Z 172,A 152.803,B 8.8704,C 0.1719,E1 8.7313,E2 298.7868} C_DIS
LIN {X -119.0496,Y 67.6051,Z 172,A 151.0312,B 8.8704,C 0.1694,E1 8.7338,E2 300.5699} C_DIS
LIN {X -116.8367,Y 71.3613,Z 172,A 149.178,B 8.8706,C 0.1653,E1 8.7364,E2 302.4247} C_DIS
LIN {X -114.6865,Y 74.768,Z 172,A 147.5023,B 8.8706,C 0.1609,E1 8.739,E2 304.0975} C_DIS
LIN {X -112.2268,Y 78.4117,Z 172,A 145.7008,B 8.8707,C 0.1559,E1 8.7418,E2 305.8924} C_DIS
LIN {X -109.9696,Y 81.5471,Z 172,A 143.9589,B 8.8707,C 0.1541,E1 8.7447,E2 307.6479} C_DIS
LIN {X -107.2855,Y 85.0474,Z 172,A 142.0868,B 8.8708,C 0.1503,E1 8.7479,E2 309.5212} C_DIS
LIN {X -104.4847,Y 88.4658,Z 172,A 140.2124,B 8.8709,C 0.1465,E1 8.7513,E2 311.3969} C_DIS
LIN {X -101.6868,Y 91.6688,Z 172,A 138.5114,B 8.8709,C 0.1413,E1 8.7544,E2 313.0865} C_DIS
LIN {X -99.2808,Y 94.2693,Z 172,A 136.9061,B 8.871,C 0.1402,E1 8.7575,E2 314.7052} C_DIS
LIN {X -96.1789,Y 97.432,Z 172,A 135.089,B 8.871,C 0.1357,E1 8.761,E2 316.5161} C_DIS
LIN {X -93.1027,Y 100.375,Z 172,A 133.3361,B 8.8711,C 0.1316,E1 8.7646,E2 318.2638} C_DIS
LIN {X -90.2164,Y 102.977,Z 172,A 131.584,B 8.8711,C 0.1305,E1 8.7683,E2 320.0295} C_DIS
LIN {X -86.8432,Y 105.8372,Z 172,A 129.7134,B 8.8711,C 0.1274,E1 8.7723,E2 321.9007} C_DIS
LIN {X -83.3849,Y 108.5827,Z 172,A 127.8467,B 8.8712,C 0.1244,E1 8.7764,E2 323.768} C_DIS
LIN {X -79.9867,Y 111.1103,Z 172,A 126.1587,B 8.8712,C 0.1199,E1 8.7802,E2 325.4442} C_DIS
LIN {X -76.9697,Y 113.2207,Z 172,A 124.501,B 8.8713,C 0.1193,E1 8.784,E2 327.1146} C_DIS
LIN {X -73.4731,Y 115.5207,Z 172,A 122.833,B 8.8713,C 0.1151,E1 8.7879,E2 328.771} C_DIS
LIN {X -70.3235,Y 117.4643,Z 172,A 121.1746,B 8.8713,C 0.1146,E1 8.7919,E2 330.4413} C_DIS
LIN {X -66.7,Y 119.5595,Z 172,A 119.4705,B 8.8714,C 0.1112,E1 8.796,E2 332.1382} C_DIS
LIN {X -62.8804,Y 121.6118,Z 172,A 117.6817,B 8.8714,C 0.1082,E1 8.8004,E2 333.9223} C_DIS
LIN {X -59.7927,Y 123.1593,Z 172,A 116.2267,B 8.8714,C 0.1065,E1 8.8041,E2 335.3774} C_DIS
LIN {X -56.6803,Y 124.6223,Z 172,A 114.7784,B 8.8714,C 0.1049,E1 8.8077,E2 336.8256} C_DIS
LIN {X -53.5465,Y 126.0006,Z 172,A 113.3373,B 8.8715,C 0.1034,E1 8.8114,E2 338.2666} C_DIS
LIN {X -50.7014,Y 127.1703,Z 172,A 112.023,B 8.8715,C 0.1024,E1 8.8148,E2 339.5831} C_DIS
LIN {X -47.2278,Y 128.5026,Z 172,A 110.4782,B 8.8715,C 0.1006,E1 8.8189,E2 341.1253} C_DIS
LIN {X -44.3587,Y 129.5192,Z 172,A 109.2214,B 8.8715,C 0.099,E1 8.8222,E2 342.379} C_DIS
LIN {X -41.2872,Y 130.5304,Z 172,A 107.8412,B 8.8715,C 0.0983,E1 8.8258,E2 343.7615} C_DIS
LIN {X -37.9813,Y 131.5308,Z 172,A 106.37,B 8.8715,C 0.0975,E1 8.8298,E2 345.2348} C_DIS
LIN {X -34.4769,Y 132.4942,Z 172,A 104.864,B 8.8715,C 0.0961,E1 8.8338,E2 346.738} C_DIS
LIN {X -31.6408,Y 133.1982,Z 172,A 103.6343,B 8.8715,C 0.0953,E1 8.8372,E2 347.9676} C_DIS
LIN {X -28.0945,Y 133.9928,Z 172,A 102.1133,B 8.8716,C 0.0944,E1 8.8413,E2 349.4878} C_DIS
LIN {X -25.2211,Y 134.5617,Z 172,A 100.8861,B 8.8716,C 0.0937,E1 8.8447,E2 350.7144} C_DIS
LIN {X -21.7387,Y 135.1695,Z 172,A 99.4039,B 8.8716,C 0.093,E1 8.8488,E2 352.1961} C_DIS
LIN {X -19.0786,Y 135.5685,Z 172,A 98.2324,B 8.8716,C 0.0933,E1 8.852,E2 353.3723} C_DIS
LIN {X -15.7366,Y 135.9976,Z 172,A 96.8675,B 8.8716,C 0.092,E1 8.8558,E2 354.731} C_DIS
LIN {X -12.6054,Y 136.3235,Z 172,A 95.5311,B 8.8716,C 0.092,E1 8.8595,E2 356.069} C_DIS
LIN {X -9.1917,Y 136.5975,Z 172,A 94.1169,B 8.8716,C 0.0912,E1 8.8634,E2 357.4802} C_DIS
LIN {X -6.1033,Y 136.7703,Z 172,A 92.8235,B 8.8716,C 0.091,E1 8.867,E2 358.7728} C_DIS
LIN {X -3.3361,Y 136.8644,Z 172,A 91.6485,B 8.8716,C 0.0912,E1 8.8703,E2 359.9492} C_DIS
LIN {X -0.2948,Y 136.9048,Z 172,A 90.3767,B 8.8716,C 0.0912,E1 8.8739,E2 361.2202} C_DIS
LIN {X 2.7427,Y 136.8776,Z 172,A 89.1026,B 8.8716,C 0.0912,E1 8.8774,E2 362.4942} C_DIS
LIN {X 5.8048,Y 136.782,Z 172,A 87.837,B 8.8716,C 0.091,E1 8.881,E2 363.7572} C_DIS
LIN {X 8.5092,Y 136.6396,Z 172,A 86.6952,B 8.8716,C 0.0913,E1 8.8841,E2 364.8995} C_DIS
LIN {X 11.9988,Y 136.3782,Z 172,A 85.2183,B 8.8716,C 0.0919,E1 8.8883,E2 366.3775} C_DIS
LIN {X 15.4311,Y 136.034,Z 172,A 83.7932,B 8.8716,C 0.0919,E1 8.8922,E2 367.7998} C_DIS
LIN {X 20.1565,Y 135.4145,Z 172,A 81.7997,B 8.8716,C 0.0926,E1 8.8977,E2 369.7925} C_DIS
LIN {X 23.0157,Y 134.9565,Z 172,A 80.5791,B 8.8716,C 0.0934,E1 8.9011,E2 371.0137} C_DIS
LIN {X 26.5022,Y 134.3168,Z 172,A 79.1074,B 8.8716,C 0.0939,E1 8.9051,E2 372.4837} C_DIS
LIN {X 29.3786,Y 133.7156,Z 172,A 77.8598,B 8.8716,C 0.095,E1 8.9085,E2 373.7331} C_DIS
LIN {X 32.312,Y 133.0364,Z 172,A 76.6191,B 8.8716,C 0.0954,E1 8.9119,E2 374.9711} C_DIS
LIN {X 35.7635,Y 132.1511,Z 172,A 75.1346,B 8.8716,C 0.0963,E1 8.9159,E2 376.4545} C_DIS
LIN {X 39.2673,Y 131.1543,Z 172,A 73.615,B 8.8716,C 0.0975,E1 8.92,E2 377.9732} C_DIS
LIN {X 42.2556,Y 130.2211,Z 172,A 72.3248,B 8.8716,C 0.0982,E1 8.9234,E2 379.2608} C_DIS
LIN {X 45.1896,Y 129.2312,Z 172,A 71.0043,B 8.8716,C 0.0999,E1 8.9269,E2 380.5841} C_DIS
LIN {X 48.5046,Y 128.0243,Z 172,A 69.5487,B 8.8716,C 0.1009,E1 8.9307,E2 382.037} C_DIS
LIN {X 51.9726,Y 126.6579,Z 172,A 67.9968,B 8.8716,C 0.1024,E1 8.9347,E2 383.5878} C_DIS
LIN {X 54.8107,Y 125.454,Z 172,A 66.7132,B 8.8716,C 0.1037,E1 8.938,E2 384.8705} C_DIS
LIN {X 57.9088,Y 124.0542,Z 172,A 65.2963,B 8.8715,C 0.1053,E1 8.9416,E2 386.2866} C_DIS
LIN {X 61.039,Y 122.5444,Z 172,A 63.8534,B 8.8715,C 0.1069,E1 8.9452,E2 387.7282} C_DIS
LIN {X 64.6767,Y 120.6653,Z 172,A 62.0597,B 8.8715,C 0.1108,E1 8.9497,E2 389.5317} C_DIS
LIN {X 68.4532,Y 118.5638,Z 172,A 60.2587,B 8.8714,C 0.1132,E1 8.9541,E2 391.3318} C_DIS
LIN {X 72.3021,Y 116.2566,Z 172,A 58.4427,B 8.8714,C 0.1147,E1 8.9584,E2 393.1405} C_DIS
LIN {X 75.649,Y 114.1078,Z 172,A 56.7986,B 8.8714,C 0.1169,E1 8.9622,E2 394.7823} C_DIS
LIN {X 79.131,Y 111.7208,Z 172,A 55.0703,B 8.8714,C 0.1189,E1 8.9662,E2 396.5061} C_DIS
LIN {X 82.5659,Y 109.2065,Z 172,A 53.2497,B 8.8713,C 0.1228,E1 8.9703,E2 398.3318} C_DIS
LIN {X 86.1581,Y 106.3956,Z 172,A 51.4353,B 8.8713,C 0.1242,E1 8.9742,E2 400.1351} C_DIS
LIN {X 89.1232,Y 103.9246,Z 172,A 49.7322,B 8.8712,C 0.129,E1 8.9779,E2 401.8494} C_DIS
LIN {X 92.4514,Y 100.9752,Z 172,A 47.8958,B 8.8712,C 0.1321,E1 8.9817,E2 403.6832} C_DIS
LIN {X 95.7224,Y 97.8797,Z 172,A 46.0372,B 8.8711,C 0.1353,E1 8.9854,E2 405.5391} C_DIS
LIN {X 98.7877,Y 94.7852,Z 172,A 44.2305,B 8.8711,C 0.1387,E1 8.9889,E2 407.3445} C_DIS
LIN {X 101.5095,Y 91.8642,Z 172,A 42.6028,B 8.871,C 0.1413,E1 8.992,E2 408.9675} C_DIS
LIN {X 104.4847,Y 88.4658,Z 172,A 40.7928,B 8.871,C 0.1437,E1 8.9953,E2 410.7684} C_DIS
LIN {X 106.8424,Y 85.6041,Z 172,A 39.2382,B 8.8709,C 0.1472,E1 8.998,E2 412.3241} C_DIS
LIN {X 109.4423,Y 82.2534,Z 172,A 37.5299,B 8.8709,C 0.1498,E1 9.0009,E2 414.0249} C_DIS
LIN {X 111.7208,Y 79.131,Z 172,A 35.8358,B 8.8708,C 0.1552,E1 9.0037,E2 415.7292} C_DIS
LIN {X 114.0131,Y 75.7909,Z 172,A 34.176,B 8.8707,C 0.1585,E1 9.0063,E2 417.3855} C_DIS
LIN {X 116.4686,Y 71.9613,Z 172,A 32.3439,B 8.8707,C 0.1616,E1 9.009,E2 419.2098} C_DIS
LIN {X 118.6173,Y 68.3607,Z 172,A 30.6378,B 8.8706,C 0.1649,E1 9.0114,E2 420.9108} C_DIS
LIN {X 120.4372,Y 65.1013,Z 172,A 29.0007,B 8.8705,C 0.1704,E1 9.0136,E2 422.5581} C_DIS
LIN {X 122.3961,Y 61.3399,Z 172,A 27.3711,B 8.8705,C 0.1718,E1 9.0156,E2 424.1708} C_DIS
LIN {X 123.7867,Y 58.4793,Z 172,A 26.0521,B 8.8704,C 0.175,E1 9.0172,E2 425.4891} C_DIS
LIN {X 125.322,Y 55.1159,Z 172,A 24.5382,B 8.8704,C 0.1783,E1 9.019,E2 427} C_DIS
LIN {X 126.5301,Y 52.2786,Z 172,A 23.2687,B 8.8703,C 0.1813,E1 9.0203,E2 428.2676} C_DIS
LIN {X 127.9089,Y 48.8128,Z 172,A 21.733,B 8.8702,C 0.1849,E1 9.0219,E2 429.8013} C_DIS
LIN {X 129.0629,Y 45.6735,Z 172,A 20.3598,B 8.8702,C 0.1881,E1 9.0232,E2 431.1722} C_DIS
LIN {X 130.0756,Y 42.7008,Z 172,A 19.0682,B 8.8701,C 0.1912,E1 9.0243,E2 432.4619} C_DIS
LIN {X 131.0594,Y 39.5775,Z 172,A 17.7353,B 8.87,C 0.1942,E1 9.0254,E2 433.7912} C_DIS
LIN {X 131.9837,Y 36.3767,Z 172,A 16.3567,B 8.87,C 0.1977,E1 9.0265,E2 435.1689} C_DIS
LIN {X 132.7709,Y 33.3866,Z 172,A 15.0288,B 8.8698,C 0.2021,E1 9.0274,E2 436.502} C_DIS
LIN {X 133.5778,Y 29.9987,Z 172,A 13.6239,B 8.8698,C 0.205,E1 9.0283,E2 437.9015} C_DIS
LIN {X 134.204,Y 27.0564,Z 172,A 12.3785,B 8.8697,C 0.2083,E1 9.029,E2 439.1463} C_DIS
LIN {X 134.8498,Y 23.6327,Z 172,A 10.9551,B 8.8696,C 0.2116,E1 9.0297,E2 440.5666} C_DIS
LIN {X 135.3669,Y 20.4641,Z 172,A 9.6542,B 8.8696,C 0.2145,E1 9.0303,E2 441.8633} C_DIS
LIN {X 135.8466,Y 17.0023,Z 172,A 8.2173,B 8.8694,C 0.2181,E1 9.0308,E2 443.2982} C_DIS
LIN {X 136.1699,Y 14.1688,Z 172,A 7.0458,B 8.8694,C 0.2211,E1 9.0311,E2 444.468} C_DIS
LIN {X 136.4462,Y 11.1936,Z 172,A 5.7812,B 8.8693,C 0.225,E1 9.0315,E2 445.7355} C_DIS
LIN {X 136.6928,Y 7.6446,Z 172,A 4.3556,B 8.8692,C 0.2279,E1 9.0317,E2 447.1545} C_DIS
LIN {X 136.8302,Y 4.5679,Z 172,A 3.091,B 8.8692,C 0.2311,E1 9.0318,E2 448.4173} C_DIS
LIN {X 136.898,Y 1.516,Z 172,A 1.9115,B 8.8691,C 0.2326,E1 9.0319,E2 449.5857} C_DIS
LIN {X 136.8984,Y -1.4662,Z 172,A 0.605,B 8.8689,C 0.2375,E1 9.0319,E2 450.9007} C_DIS
LIN {X 136.8302,Y -4.5679,Z 172,A -0.6717,B 8.8689,C 0.2408,E1 9.0318,E2 452.1759} C_DIS
LIN {X 136.7079,Y -7.345,Z 172,A -1.8188,B 8.8688,C 0.2438,E1 9.0316,E2 453.322} C_DIS
LIN {X 136.5062,Y -10.4422,Z 172,A -3.0987,B 8.8687,C 0.2472,E1 9.0314,E2 454.6008} C_DIS
LIN {X 136.2026,Y -13.8641,Z 172,A -4.5154,B 8.8686,C 0.2509,E1 9.031,E2 456.0163} C_DIS
LIN {X 135.9185,Y -16.3996,Z 172,A -5.6031,B 8.8685,C 0.2544,E1 9.0307,E2 457.1075} C_DIS
LIN {X 135.4145,Y -20.1565,Z 172,A -7.1301,B 8.8684,C 0.2577,E1 9.0301,E2 458.6286} C_DIS
LIN {X 134.9565,Y -23.0157,Z 172,A -8.3437,B 8.8683,C 0.2612,E1 9.0295,E2 459.8436} C_DIS
LIN {X 134.3168,Y -26.5022,Z 172,A -9.7861,B 8.8682,C 0.2645,E1 9.0288,E2 461.2824} C_DIS
LIN {X 133.7156,Y -29.3786,Z 172,A -11.0176,B 8.8681,C 0.2681,E1 9.028,E2 462.5153} C_DIS
LIN {X 132.9743,Y -32.5697,Z 172,A -12.3496,B 8.868,C 0.2711,E1 9.0272,E2 463.8438} C_DIS
LIN {X 132.1511,Y -35.7635,Z 172,A -13.7097,B 8.8679,C 0.2745,E1 9.0262,E2 465.2027} C_DIS
LIN {X 131.1543,Y -39.2673,Z 172,A -15.2119,B 8.8678,C 0.2783,E1 9.025,E2 466.7037} C_DIS
LIN {X 130.3008,Y -42.0062,Z 172,A -16.4092,B 8.8677,C 0.2816,E1 9.024,E2 467.9018} C_DIS
LIN {X 129.0751,Y -45.6399,Z 172,A -17.9764,B 8.8676,C 0.2852,E1 9.0226,E2 469.4659} C_DIS
LIN {X 128.0243,Y -48.5046,Z 172,A -19.2208,B 8.8675,C 0.288,E1 9.0214,E2 470.7075} C_DIS
LIN {X 126.8492,Y -51.4981,Z 172,A -20.6055,B 8.8673,C 0.2925,E1 9.02,E2 472.0985} C_DIS
LIN {X 125.454,Y -54.8107,Z 172,A -22.0372,B 8.8673,C 0.295,E1 9.0184,E2 473.5226} C_DIS
LIN {X 124.0415,Y -57.9363,Z 172,A -23.4601,B 8.8671,C 0.2986,E1 9.0167,E2 474.9455} C_DIS
LIN {X 122.5444,Y -61.039,Z 172,A -24.8816,B 8.8671,C 0.3019,E1 9.015,E2 476.3658} C_DIS
LIN {X 120.9781,Y -64.0873,Z 172,A -26.3195,B 8.8669,C 0.3058,E1 9.0131,E2 477.8058} C_DIS
LIN {X 119.0496,Y -67.6051,Z 172,A -28.0488,B 8.8667,C 0.3112,E1 9.0108,E2 479.5432} C_DIS
LIN {X 116.8367,Y -71.3613,Z 172,A -29.8487,B 8.8665,C 0.3153,E1 9.0082,E2 481.3419} C_DIS
LIN {X 114.5901,Y -74.9165,Z 172,A -31.5298,B 8.8665,C 0.318,E1 9.0056,E2 483.0149} C_DIS
LIN {X 112.2268,Y -78.4117,Z 172,A -33.2293,B 8.8663,C 0.3208,E1 9.003,E2 484.7078} C_DIS
LIN {X 109.9696,Y -81.5471,Z 172,A -34.9234,B 8.8661,C 0.3264,E1 9.0002,E2 486.4133} C_DIS
LIN {X 107.2855,Y -85.0474,Z 172,A -36.7458,B 8.8661,C 0.3302,E1 8.997,E2 488.2346} C_DIS
LIN {X 104.4847,Y -88.4658,Z 172,A -38.5717,B 8.8659,C 0.334,E1 8.9938,E2 490.0594} C_DIS
LIN {X 101.6868,Y -91.6688,Z 172,A -40.2302,B 8.8659,C 0.3353,E1 8.9907,E2 491.7043} C_DIS
LIN {X 99.2808,Y -94.2693,Z 172,A -41.8072,B 8.8656,C 0.3406,E1 8.9877,E2 493.2947} C_DIS
LIN {X 96.2717,Y -97.3398,Z 172,A -43.5296,B 8.8656,C 0.3428,E1 8.9843,E2 495.0093} C_DIS
LIN {X 93.1027,Y -100.375,Z 172,A -45.2866,B 8.8655,C 0.3449,E1 8.9808,E2 496.7579} C_DIS
LIN {X 90.346,Y -102.8638,Z 172,A -46.8231,B 8.8653,C 0.3476,E1 8.9776,E2 498.2937} C_DIS
LIN {X 87.3417,Y -105.4259,Z 172,A -48.5278,B 8.8652,C 0.352,E1 8.9739,E2 500.0066} C_DIS
LIN {X 84.0831,Y -108.043,Z 172,A -50.2853,B 8.865,C 0.3554,E1 8.97,E2 501.7669} C_DIS
LIN {X 80.561,Y -110.694,Z 172,A -52.1091,B 8.865,C 0.3583,E1 8.966,E2 503.5898} C_DIS
LIN {X 77.106,Y -113.1284,Z 172,A -53.8363,B 8.8648,C 0.3605,E1 8.962,E2 505.3133} C_DIS
LIN {X 73.4439,Y -115.5395,Z 172,A -55.5782,B 8.8648,C 0.3616,E1 8.9579,E2 507.0451} C_DIS
LIN {X 70.3235,Y -117.4643,Z 172,A -57.1953,B 8.8646,C 0.3659,E1 8.954,E2 508.674} C_DIS
LIN {X 66.7,Y -119.5595,Z 172,A -58.8324,B 8.8646,C 0.3661,E1 8.9501,E2 510.2981} C_DIS
LIN {X 63.2319,Y -121.4272,Z 172,A -60.493,B 8.8645,C 0.3688,E1 8.946,E2 511.9616} C_DIS
LIN {X 59.7927,Y -123.1593,Z 172,A -62.0632,B 8.8645,C 0.3702,E1 8.9421,E2 513.5279} C_DIS
LIN {X 56.6803,Y -124.6223,Z 172,A -63.4902,B 8.8644,C 0.3718,E1 8.9385,E2 514.9546} C_DIS
LIN {X 53.8428,Y -125.8725,Z 172,A -64.7668,B 8.8644,C 0.373,E1 8.9352,E2 516.2295} C_DIS
LIN {X 50.7014,Y -127.1703,Z 172,A -66.2081,B 8.8642,C 0.3751,E1 8.9315,E2 517.6743} C_DIS
LIN {X 47.2278,Y -128.5026,Z 172,A -67.7337,B 8.8642,C 0.3762,E1 8.9275,E2 519.1971} C_DIS
LIN {X 44.3587,Y -129.5192,Z 172,A -69.0176,B 8.8642,C 0.3778,E1 8.9241,E2 520.4833} C_DIS
LIN {X 41.1728,Y -130.567,Z 172,A -70.3912,B 8.8641,C 0.3786,E1 8.9204,E2 521.8541} C_DIS
LIN {X 37.9813,Y -131.5308,Z 172,A -71.7968,B 8.8641,C 0.3801,E1 8.9167,E2 523.262} C_DIS
LIN {X 34.4769,Y -132.4942,Z 172,A -73.2887,B 8.864,C 0.3809,E1 8.9127,E2 524.7513} C_DIS
LIN {X 31.6112,Y -133.2053,Z 172,A -74.5179,B 8.864,C 0.3817,E1 8.9093,E2 525.9804} C_DIS
LIN {X 28.6124,Y -133.881,Z 172,A -75.8439,B 8.8639,C 0.3835,E1 8.9057,E2 527.3123} C_DIS
LIN {X 25.2211,Y -134.5617,Z 172,A -77.2353,B 8.8639,C 0.3833,E1 8.9019,E2 528.6976} C_DIS
LIN {X 21.7387,Y -135.1695,Z 172,A -78.7081,B 8.8639,C 0.3841,E1 8.8978,E2 530.1705} C_DIS
LIN {X 18.8846,Y -135.5963,Z 172,A -79.9282,B 8.8639,C 0.3849,E1 8.8945,E2 531.3928} C_DIS
LIN {X 15.7366,Y -135.9976,Z 172,A -81.2039,B 8.8639,C 0.3845,E1 8.8909,E2 532.6626} C_DIS
LIN {X 12.6054,Y -136.3235,Z 172,A -82.5622,B 8.8638,C 0.3859,E1 8.8871,E2 534.0268} C_DIS
LIN {X 9.1917,Y -136.5975,Z 172,A -83.9718,B 8.8638,C 0.3859,E1 8.8832,E2 535.4343} C_DIS
LIN {X 6.1033,Y -136.7703,Z 172,A -85.2619,B 8.8638,C 0.3862,E1 8.8796,E2 536.7246} C_DIS
LIN {X 3.3361,Y -136.8644,Z 172,A -86.4348,B 8.8638,C 0.3867,E1 8.8763,E2 537.8997} C_DIS
LIN {X 0.9853,Y -136.901,Z 172,A -87.2015,B 8.8639,C 0.3826,E1 8.8743,E2 538.6393} C_DIS
Enddeposition()
LIN {X 0.9853,Y -136.901,Z 172,A -87.2015,B 8.8639,C 0.3826,E1 8.8743,E2 538.6393} C_DIS
Startdeposition()
$VEL.CP = VEL_PRINT
LIN {X 2.6432,Y -137.7886,Z 172,A -86.0756,B 8.7909,C 0.3805,E1 8.8044,E2 537.5121} C_DIS
LIN {X 6.7424,Y -137.6485,Z 172,A -84.3438,B 8.7909,C 0.3795,E1 8.8092,E2 535.7761} C_DIS
LIN {X 10.7154,Y -137.3979,Z 172,A -82.4375,B 8.7912,C 0.3739,E1 8.8146,E2 533.8364} C_DIS
LIN {X 15.9931,Y -136.8826,Z 172,A -79.835,B 8.7915,C 0.3648,E1 8.822,E2 531.1807} C_DIS
LIN {X 21.2926,Y -136.1586,Z 172,A -78.3423,B 8.791,C 0.3785,E1 8.8258,E2 529.7818} C_DIS
LIN {X 24.5978,Y -135.6006,Z 172,A -76.8822,B 8.791,C 0.3763,E1 8.8299,E2 528.3122} C_DIS
LIN {X 27.5597,Y -135.0294,Z 172,A -75.6343,B 8.791,C 0.3756,E1 8.8333,E2 527.0643} C_DIS
LIN {X 30.84,Y -134.3182,Z 172,A -74.2653,B 8.7911,C 0.3751,E1 8.837,E2 525.6978} C_DIS
LIN {X 34.7545,Y -133.3611,Z 172,A -72.6206,B 8.7911,C 0.3743,E1 8.8415,E2 524.056} C_DIS
LIN {X 39.1231,Y -132.1438,Z 172,A -70.668,B 8.7913,C 0.3712,E1 8.8467,E2 522.0932} C_DIS
LIN {X 45.0435,Y -130.2441,Z 172,A -68.0685,B 8.7913,C 0.3683,E1 8.8536,E2 519.49} C_DIS
LIN {X 52.4207,Y -127.456,Z 172,A -64.3841,B 8.7919,C 0.3559,E1 8.8634,E2 515.7504} C_DIS
LIN {X 56.4257,Y -125.7321,Z 172,A -63.0241,B 8.7916,C 0.3632,E1 8.8667,E2 514.4478} C_DIS
LIN {X 59.684,Y -124.2188,Z 172,A -61.5628,B 8.7916,C 0.3618,E1 8.8704,E2 512.9895} C_DIS
LIN {X 62.7264,Y -122.7104,Z 172,A -60.2047,B 8.7916,C 0.361,E1 8.8737,E2 511.6372} C_DIS
LIN {X 65.9657,Y -121.002,Z 172,A -58.6392,B 8.7918,C 0.3578,E1 8.8776,E2 510.0649} C_DIS
LIN {X 69.5424,Y -118.9827,Z 172,A -56.6827,B 8.7921,C 0.3499,E1 8.8824,E2 508.0746} C_DIS
LIN {X 72.5323,Y -117.1841,Z 172,A -55.4484,B 8.7921,C 0.3522,E1 8.8853,E2 506.867} C_DIS
LIN {X 76.3177,Y -114.7546,Z 172,A -53.5966,B 8.7921,C 0.3494,E1 8.8896,E2 505.016} C_DIS
LIN {X 80.637,Y -111.7618,Z 172,A -50.7906,B 8.7928,C 0.332,E1 8.8962,E2 502.1269} C_DIS
LIN {X 85.3505,Y -108.205,Z 172,A -49.2988,B 8.7922,C 0.3484,E1 8.8992,E2 500.7582} C_DIS
LIN {X 91.8014,Y -102.7886,Z 172,A -45.7853,B 8.7925,C 0.3414,E1 8.9067,E2 497.24} C_DIS
LIN {X 97.241,Y -97.6583,Z 172,A -42.8749,B 8.7925,C 0.3393,E1 8.9126,E2 494.3524} C_DIS
LIN {X 101.533,Y -93.188,Z 172,A -40.1875,B 8.7928,C 0.3313,E1 8.9178,E2 491.6483} C_DIS
LIN {X 104.2269,Y -90.1653,Z 172,A -38.584,B 8.7929,C 0.3293,E1 8.9207,E2 490.0534} C_DIS
LIN {X 107.3523,Y -86.4201,Z 172,A -36.0578,B 8.7935,C 0.3136,E1 8.9253,E2 487.4607} C_DIS
LIN {X 109.5074,Y -83.6725,Z 172,A -35.0046,B 8.7933,C 0.319,E1 8.927,E2 486.4577} C_DIS
LIN {X 111.8171,Y -80.5607,Z 172,A -33.2844,B 8.7935,C 0.3127,E1 8.9299,E2 484.7218} C_DIS
LIN {X 114.0674,Y -77.3406,Z 172,A -31.715,B 8.7936,C 0.3101,E1 8.9324,E2 483.159} C_DIS
LIN {X 117.8739,Y -71.4051,Z 172,A -29.0238,B 8.7936,C 0.3082,E1 8.9364,E2 480.4957} C_DIS
LIN {X 119.3714,Y -68.8727,Z 172,A -27.6226,B 8.7939,C 0.3011,E1 8.9383,E2 479.0704} C_DIS
LIN {X 121.2854,Y -65.4436,Z 172,A -25.9593,B 8.7941,C 0.2961,E1 8.9406,E2 477.4014} C_DIS
LIN {X 122.8971,Y -62.3597,Z 172,A -24.7347,B 8.7941,C 0.2973,E1 8.9421,E2 476.2038} C_DIS
LIN {X 125.6508,Y -56.6075,Z 172,A -22.1851,B 8.7942,C 0.2926,E1 8.9452,E2 473.6647} C_DIS
LIN {X 126.7932,Y -54.0041,Z 172,A -20.8535,B 8.7944,C 0.286,E1 8.9467,E2 472.3127} C_DIS
LIN {X 128.0314,Y -50.997,Z 172,A -19.2876,B 8.7947,C 0.2775,E1 8.9483,E2 470.7179} C_DIS
LIN {X 129.3455,Y -47.5693,Z 172,A -18.0168,B 8.7947,C 0.2791,E1 8.9495,E2 469.4785} C_DIS
LIN {X 130.2529,Y -45.0179,Z 172,A -16.9237,B 8.7947,C 0.2767,E1 8.9505,E2 468.3883} C_DIS
LIN {X 131.2807,Y -41.9261,Z 172,A -15.5558,B 8.7948,C 0.2726,E1 8.9517,E2 467.0173} C_DIS
LIN {X 132.4204,Y -38.1785,Z 172,A -14.0046,B 8.7949,C 0.2698,E1 8.9529,E2 465.4744} C_DIS
LIN {X 133.1877,Y -35.4046,Z 172,A -12.7713,B 8.7951,C 0.2656,E1 8.9538,E2 464.2351} C_DIS
LIN {X 134.0078,Y -32.162,Z 172,A -11.3726,B 8.7951,C 0.2615,E1 8.9548,E2 462.8339} C_DIS
LIN {X 134.9028,Y -28.1818,Z 172,A -9.4861,B 8.7955,C 0.2523,E1 8.9559,E2 460.9214} C_DIS
LIN {X 136.184,Y -21.1283,Z 172,A -6.3849,B 8.7958,C 0.241,E1 8.9573,E2 457.8015} C_DIS
LIN {X 136.7691,Y -16.9445,Z 172,A -5.1786,B 8.7956,C 0.2484,E1 8.9578,E2 456.6642} C_DIS
LIN {X 137.4814,Y -9.5717,Z 172,A -2.5436,B 8.7956,C 0.2496,E1 8.9585,E2 454.0831} C_DIS
LIN {X 137.7847,Y -2.8755,Z 172,A 0.5772,B 8.796,C 0.234,E1 8.9589,E2 450.9175} C_DIS
LIN {X 137.7425,Y 4.4657,Z 172,A 3.9149,B 8.7963,C 0.2187,E1 8.9587,E2 447.5408} C_DIS
LIN {X 137.3883,Y 10.8419,Z 172,A 6.2544,B 8.7963,C 0.2182,E1 8.9583,E2 445.2392} C_DIS
LIN {X 137.0744,Y 14.2601,Z 172,A 7.7828,B 8.7965,C 0.2118,E1 8.9579,E2 443.6966} C_DIS
LIN {X 136.6077,Y 18.191,Z 172,A 9.3175,B 8.7965,C 0.2095,E1 8.9573,E2 442.1746} C_DIS
LIN {X 136.0096,Y 22.2283,Z 172,A 11.1138,B 8.7967,C 0.2025,E1 8.9565,E2 440.3642} C_DIS
LIN {X 135.2205,Y 26.6167,Z 172,A 13.0206,B 8.7969,C 0.196,E1 8.9555,E2 438.4491} C_DIS
LIN {X 134.3504,Y 30.6992,Z 172,A 14.5709,B 8.7969,C 0.1953,E1 8.9546,E2 436.921} C_DIS
LIN {X 133.5199,Y 34.1315,Z 172,A 15.934,B 8.7969,C 0.1935,E1 8.9537,E2 435.5701} C_DIS
LIN {X 132.6673,Y 37.3078,Z 172,A 17.3173,B 8.797,C 0.1894,E1 8.9527,E2 434.1837} C_DIS
LIN {X 131.7853,Y 40.3121,Z 172,A 18.5992,B 8.797,C 0.1862,E1 8.9516,E2 432.9033} C_DIS
LIN {X 130.7023,Y 43.6962,Z 172,A 20.0377,B 8.7972,C 0.183,E1 8.9504,E2 431.4687} C_DIS
LIN {X 129.4994,Y 47.1434,Z 172,A 21.4905,B 8.7972,C 0.1803,E1 8.949,E2 430.023} C_DIS
LIN {X 128.1753,Y 50.6367,Z 172,A 23.2519,B 8.7974,C 0.1715,E1 8.9472,E2 428.2342} C_DIS
LIN {X 126.8686,Y 53.8271,Z 172,A 24.4607,B 8.7974,C 0.1727,E1 8.946,E2 427.053} C_DIS
LIN {X 125.6127,Y 56.6927,Z 172,A 25.7562,B 8.7974,C 0.1694,E1 8.9445,E2 425.7572} C_DIS
LIN {X 124.0672,Y 60.0013,Z 172,A 27.2354,B 8.7974,C 0.1664,E1 8.9427,E2 424.282} C_DIS
LIN {X 122.4352,Y 63.2669,Z 172,A 28.8904,B 8.7976,C 0.1594,E1 8.9406,E2 422.6088} C_DIS
LIN {X 120.1949,Y 67.4251,Z 172,A 30.7467,B 8.7976,C 0.1569,E1 8.9381,E2 420.7649} C_DIS
LIN {X 117.8279,Y 71.4812,Z 172,A 32.6422,B 8.7977,C 0.1533,E1 8.9354,E2 418.8755} C_DIS
LIN {X 115.7218,Y 74.843,Z 172,A 34.3494,B 8.7978,C 0.148,E1 8.9328,E2 417.1601} C_DIS
LIN {X 113.2468,Y 78.5375,Z 172,A 36.1286,B 8.7978,C 0.1452,E1 8.9301,E2 415.3888} C_DIS
LIN {X 110.7256,Y 82.0541,Z 172,A 37.9611,B 8.7979,C 0.1402,E1 8.927,E2 413.5512} C_DIS
LIN {X 108.006,Y 85.6022,Z 172,A 39.7854,B 8.7979,C 0.1368,E1 8.9239,E2 411.7304} C_DIS
LIN {X 105.0785,Y 89.171,Z 172,A 41.6496,B 8.798,C 0.1337,E1 8.9206,E2 409.8722} C_DIS
LIN {X 102.1692,Y 92.4901,Z 172,A 43.9673,B 8.7982,C 0.1194,E1 8.9161,E2 407.4929} C_DIS
LIN {X 98.7511,Y 96.1316,Z 172,A 45.5487,B 8.7982,C 0.1258,E1 8.9132,E2 405.9733} C_DIS
LIN {X 94.9155,Y 99.9208,Z 172,A 47.6917,B 8.7982,C 0.1234,E1 8.9089,E2 403.8421} C_DIS
LIN {X 92.0336,Y 102.5806,Z 172,A 49.3452,B 8.7982,C 0.1198,E1 8.9055,E2 402.1852} C_DIS
LIN {X 88.8457,Y 105.3542,Z 172,A 51.1034,B 8.7982,C 0.1165,E1 8.9018,E2 400.4264} C_DIS
LIN {X 85.5295,Y 108.0638,Z 172,A 52.863,B 8.7983,C 0.1138,E1 8.8979,E2 398.669} C_DIS
LIN {X 81.9219,Y 110.8238,Z 172,A 54.962,B 8.7984,C 0.1061,E1 8.8932,E2 396.5433} C_DIS
LIN {X 79.0322,Y 112.9026,Z 172,A 56.0283,B 8.7984,C 0.1123,E1 8.8909,E2 395.5285} C_DIS
LIN {X 76.3922,Y 114.7048,Z 172,A 57.3782,B 8.7984,C 0.1098,E1 8.8877,E2 394.1759} C_DIS
LIN {X 73.2333,Y 116.7475,Z 172,A 59.0394,B 8.7984,C 0.1053,E1 8.8838,E2 392.5023} C_DIS
LIN {X 69.6151,Y 118.94,Z 172,A 60.7768,B 8.7984,C 0.1032,E1 8.8796,E2 390.7675} C_DIS
LIN {X 65.6336,Y 121.1831,Z 172,A 62.7094,B 8.7984,C 0.0999,E1 8.8749,E2 388.8307} C_DIS
LIN {X 60.6217,Y 123.7641,Z 172,A 64.9495,B 8.7984,C 0.099,E1 8.8693,E2 386.6035} C_DIS
LIN {X 57.4828,Y 125.2528,Z 172,A 66.3485,B 8.7984,C 0.0982,E1 8.8658,E2 385.2102} C_DIS
LIN {X 53.767,Y 126.8937,Z 172,A 67.9714,B 8.7985,C 0.0977,E1 8.8617,E2 383.5957} C_DIS
LIN {X 51.1031,Y 127.9886,Z 172,A 69.1936,B 8.7985,C 0.0959,E1 8.8585,E2 382.3704} C_DIS
LIN {X 48.0159,Y 129.1782,Z 172,A 70.5703,B 8.7985,C 0.0945,E1 8.8549,E2 380.9937} C_DIS
LIN {X 44.9982,Y 130.2598,Z 172,A 71.9004,B 8.7985,C 0.0933,E1 8.8514,E2 379.6641} C_DIS
LIN {X 41.8061,Y 131.3191,Z 172,A 73.2894,B 8.7985,C 0.0922,E1 8.8477,E2 378.2764} C_DIS
LIN {X 38.1883,Y 132.4175,Z 172,A 74.8498,B 8.7985,C 0.0912,E1 8.8435,E2 376.7178} C_DIS
LIN {X 34.9426,Y 133.3109,Z 172,A 76.3971,B 8.7986,C 0.0872,E1 8.8393,E2 375.1524} C_DIS
LIN {X 28.7234,Y 134.7871,Z 172,A 78.9234,B 8.7986,C 0.0882,E1 8.8325,E2 372.6431} C_DIS
LIN {X 25.7042,Y 135.395,Z 172,A 80.1987,B 8.7986,C 0.0876,E1 8.829,E2 371.3687} C_DIS
LIN {X 21.7484,Y 136.088,Z 172,A 82.2054,B 8.7986,C 0.0802,E1 8.8234,E2 369.3206} C_DIS
LIN {X 18.2225,Y 136.6036,Z 172,A 83.2259,B 8.7986,C 0.0887,E1 8.8207,E2 368.3579} C_DIS
LIN {X 12.8227,Y 137.216,Z 172,A 85.7194,B 8.7986,C 0.0835,E1 8.8137,E2 365.8362} C_DIS
LIN {X 9.6985,Y 137.4721,Z 172,A 87.743,B 8.7988,C 0.0693,E1 8.8078,E2 363.7231} C_DIS
LIN {X 3.3028,Y 137.7749,Z 172,A 89.4391,B 8.7986,C 0.0877,E1 8.8034,E2 362.1488} C_DIS
LIN {X -3.0847,Y 137.7809,Z 172,A 92.1587,B 8.7986,C 0.0866,E1 8.7958,E2 359.4227} C_DIS
LIN {X -11.2681,Y 137.3523,Z 172,A 95.6757,B 8.7986,C 0.0852,E1 8.786,E2 355.894} C_DIS
LIN {X -16.5075,Y 136.8212,Z 172,A 97.6691,B 8.7986,C 0.0896,E1 8.7805,E2 353.9261} C_DIS
LIN {X -19.3426,Y 136.4492,Z 172,A 99.3726,B 8.7986,C 0.0805,E1 8.7756,E2 352.1593} C_DIS
LIN {X -23.0729,Y 135.8686,Z 172,A 100.6171,B 8.7986,C 0.0874,E1 8.7723,E2 350.9563} C_DIS
LIN {X -26.5968,Y 135.2243,Z 172,A 102.0407,B 8.7986,C 0.0894,E1 8.7684,E2 349.5418} C_DIS
LIN {X -30.0534,Y 134.4979,Z 172,A 103.4631,B 8.7986,C 0.0912,E1 8.7645,E2 348.126} C_DIS
LIN {X -32.3746,Y 133.9565,Z 172,A 104.5351,B 8.7986,C 0.0904,E1 8.7616,E2 347.0445} C_DIS
LIN {X -36.2887,Y 132.9519,Z 172,A 106.2007,B 8.7986,C 0.0919,E1 8.7571,E2 345.382} C_DIS
LIN {X -40.603,Y 131.6963,Z 172,A 108.0942,B 8.7986,C 0.093,E1 8.752,E2 343.4866} C_DIS
LIN {X -43.8871,Y 130.6387,Z 172,A 109.9672,B 8.7986,C 0.0865,E1 8.7469,E2 341.5601} C_DIS
LIN {X -47.7294,Y 129.2855,Z 172,A 111.1683,B 8.7986,C 0.097,E1 8.744,E2 340.4215} C_DIS
LIN {X -50.7293,Y 128.1393,Z 172,A 112.5874,B 8.7986,C 0.097,E1 8.7402,E2 338.993} C_DIS
LIN {X -55.0792,Y 126.3284,Z 172,A 114.6708,B 8.7986,C 0.097,E1 8.7348,E2 336.8957} C_DIS
LIN {X -58.3389,Y 124.857,Z 172,A 116.0843,B 8.7985,C 0.1001,E1 8.7313,E2 335.4925} C_DIS
LIN {X -62.0952,Y 123.0317,Z 172,A 117.6671,B 8.7985,C 0.1051,E1 8.7274,E2 333.9301} C_DIS
LIN {X -64.392,Y 121.8449,Z 172,A 118.9054,B 8.7985,C 0.1037,E1 8.7242,E2 332.6725} C_DIS
LIN {X -69.4277,Y 119.0501,Z 172,A 121.3565,B 8.7985,C 0.1062,E1 8.7183,E2 330.2164} C_DIS
LIN {X -73.1391,Y 116.8065,Z 172,A 123.2049,B 8.7984,C 0.1082,E1 8.7139,E2 328.364} C_DIS
LIN {X -76.7638,Y 114.4568,Z 172,A 125.0441,B 8.7984,C 0.1103,E1 8.7096,E2 326.521} C_DIS
LIN {X -80.3377,Y 111.977,Z 172,A 126.8557,B 8.7984,C 0.1134,E1 8.7054,E2 324.7107} C_DIS
LIN {X -84.64,Y 108.7616,Z 172,A 128.8241,B 8.7982,C 0.1218,E1 8.7011,E2 322.7771} C_DIS
LIN {X -88.2221,Y 105.8772,Z 172,A 131.0304,B 8.7982,C 0.1204,E1 8.6963,E2 320.5362} C_DIS
LIN {X -91.4226,Y 103.1256,Z 172,A 132.8399,B 8.7982,C 0.1228,E1 8.6925,E2 318.7215} C_DIS
LIN {X -95.0478,Y 99.7943,Z 172,A 134.9127,B 8.7982,C 0.1265,E1 8.6882,E2 316.6474} C_DIS
LIN {X -98.2106,Y 96.6834,Z 172,A 136.7233,B 8.7981,C 0.1309,E1 8.6847,E2 314.8429} C_DIS
LIN {X -100.8528,Y 93.9237,Z 172,A 138.4005,B 8.7981,C 0.1328,E1 8.6814,E2 313.1561} C_DIS
LIN {X -103.877,Y 90.5678,Z 172,A 140.2593,B 8.798,C 0.1372,E1 8.678,E2 311.3016} C_DIS
LIN {X -106.6685,Y 87.2627,Z 172,A 142.0128,B 8.798,C 0.142,E1 8.6749,E2 309.5555} C_DIS
LIN {X -111.3826,Y 81.1602,Z 172,A 145.3802,B 8.7978,C 0.1469,E1 8.6692,E2 306.1714} C_DIS
LIN {X -113.9457,Y 77.5205,Z 172,A 147.2605,B 8.7978,C 0.1508,E1 8.6662,E2 304.2893} C_DIS
LIN {X -116.648,Y 73.391,Z 172,A 149.1455,B 8.7976,C 0.1586,E1 8.6634,E2 302.4272} C_DIS
LIN {X -118.357,Y 70.6015,Z 172,A 151.488,B 8.7978,C 0.1458,E1 8.6599,E2 299.963} C_DIS
LIN {X -121.5631,Y 64.9268,Z 172,A 153.3451,B 8.7975,C 0.1668,E1 8.6575,E2 298.2158} C_DIS
LIN {X -122.9853,Y 62.1864,Z 172,A 154.6335,B 8.7975,C 0.1701,E1 8.6559,E2 296.9281} C_DIS
LIN {X -124.6087,Y 58.8679,Z 172,A 156.1775,B 8.7973,C 0.174,E1 8.654,E2 295.3847} C_DIS
LIN {X -125.9295,Y 55.9844,Z 172,A 157.5934,B 8.7973,C 0.1759,E1 8.6524,E2 293.9579} C_DIS
LIN {X -127.2804,Y 52.8411,Z 172,A 158.9787,B 8.7973,C 0.1803,E1 8.6509,E2 292.5787} C_DIS
LIN {X -128.5163,Y 49.7594,Z 172,A 160.4706,B 8.7972,C 0.1823,E1 8.6494,E2 291.0744} C_DIS
LIN {X -130.2314,Y 45.08,Z 172,A 162.5456,B 8.797,C 0.1879,E1 8.6474,E2 289.001} C_DIS
LIN {X -131.4132,Y 41.5114,Z 172,A 164.2237,B 8.797,C 0.1904,E1 8.646,E2 287.3102} C_DIS
LIN {X -132.6726,Y 37.2888,Z 172,A 166.0059,B 8.7969,C 0.1963,E1 8.6446,E2 285.536} C_DIS
LIN {X -133.7499,Y 33.2252,Z 172,A 167.7007,B 8.7967,C 0.2021,E1 8.6434,E2 283.8498} C_DIS
LIN {X -134.346,Y 30.7182,Z 172,A 168.7947,B 8.7967,C 0.2048,E1 8.6427,E2 282.754} C_DIS
LIN {X -135.2169,Y 26.6355,Z 172,A 170.5468,B 8.7966,C 0.2095,E1 8.6417,E2 281.0016} C_DIS
LIN {X -135.8151,Y 23.3941,Z 172,A 171.9221,B 8.7965,C 0.2133,E1 8.6411,E2 279.627} C_DIS
LIN {X -136.5341,Y 18.7487,Z 172,A 173.9447,B 8.7964,C 0.2179,E1 8.6402,E2 277.5978} C_DIS
LIN {X -137.0053,Y 14.9023,Z 172,A 175.6072,B 8.7963,C 0.2217,E1 8.6397,E2 275.9303} C_DIS
LIN {X -137.3618,Y 11.1561,Z 172,A 177.3597,B 8.7963,C 0.2232,E1 8.6393,E2 274.1557} C_DIS
LIN {X -137.6094,Y 7.5208,Z 172,A 178.7996,B 8.7961,C 0.2288,E1 8.639,E2 272.7267} C_DIS
LIN {X -137.7636,Y 3.7078,Z 172,A -179.6342,B 8.796,C 0.2337,E1 8.6389,E2 271.1646} C_DIS
LIN {X -137.8131,Y -0.6785,Z 172,A -177.7118,B 8.7959,C 0.2374,E1 8.6389,E2 269.2315} C_DIS
LIN {X -137.7204,Y -5.0719,Z 172,A -175.883,B 8.7957,C 0.2427,E1 8.639,E2 267.4041} C_DIS
LIN {X -137.5036,Y -9.2673,Z 172,A -174.0382,B 8.7957,C 0.2461,E1 8.6393,E2 265.5485} C_DIS
LIN {X -137.1103,Y -13.9208,Z 172,A -172.2351,B 8.7954,C 0.2539,E1 8.6398,E2 263.7646} C_DIS
LIN {X -136.7433,Y -17.1565,Z 172,A -170.8302,B 8.7954,C 0.257,E1 8.6402,E2 262.3544} C_DIS
LIN {X -136.2263,Y -20.8555,Z 172,A -169.1763,B 8.7952,C 0.2598,E1 8.6409,E2 260.689} C_DIS
LIN {X -135.6716,Y -24.2013,Z 172,A -167.7805,B 8.7952,C 0.264,E1 8.6416,E2 259.2962} C_DIS
LIN {X -135.0173,Y -27.6193,Z 172,A -166.3334,B 8.795,C 0.2681,E1 8.6424,E2 257.8503} C_DIS
LIN {X -134.2951,Y -30.9412,Z 172,A -164.8976,B 8.7949,C 0.2717,E1 8.6432,E2 256.4127} C_DIS
LIN {X -133.3677,Y -34.7298,Z 172,A -163.1068,B 8.7949,C 0.2735,E1 8.6445,E2 254.6019} C_DIS
LIN {X -132.2199,Y -38.8632,Z 172,A -161.4115,B 8.7946,C 0.2799,E1 8.6458,E2 252.919} C_DIS
LIN {X -131.0285,Y -42.7159,Z 172,A -159.4593,B 8.7946,C 0.2799,E1 8.6475,E2 250.9332} C_DIS
LIN {X -129.4701,Y -47.2249,Z 172,A -157.6949,B 8.7943,C 0.2889,E1 8.6491,E2 249.198} C_DIS
LIN {X -127.8414,Y -51.4683,Z 172,A -155.7622,B 8.7942,C 0.2932,E1 8.6511,E2 247.2611} C_DIS
LIN {X -126.4109,Y -54.8884,Z 172,A -154.2301,B 8.7941,C 0.2974,E1 8.6527,E2 245.7312} C_DIS
LIN {X -124.738,Y -58.5962,Z 172,A -152.5136,B 8.7939,C 0.3014,E1 8.6547,E2 244.0127} C_DIS
LIN {X -123.4422,Y -61.2741,Z 172,A -151.2247,B 8.7939,C 0.3037,E1 8.6563,E2 242.7179} C_DIS
LIN {X -120.6208,Y -66.6601,Z 172,A -148.8848,B 8.7935,C 0.3132,E1 8.6594,E2 240.4034} C_DIS
LIN {X -119.0515,Y -69.4253,Z 172,A -147.2938,B 8.7935,C 0.312,E1 8.6616,E2 238.7791} C_DIS
LIN {X -116.831,Y -73.0997,Z 172,A -145.4537,B 8.7935,C 0.3153,E1 8.6643,E2 236.9329} C_DIS
LIN {X -114.538,Y -76.6421,Z 172,A -143.6795,B 8.7933,C 0.3192,E1 8.6671,E2 235.1571} C_DIS
LIN {X -111.9311,Y -80.4018,Z 172,A -141.735,B 8.7932,C 0.3228,E1 8.6702,E2 233.2081} C_DIS
LIN {X -109.2111,Y -84.0598,Z 172,A -139.8247,B 8.793,C 0.3268,E1 8.6734,E2 231.2968} C_DIS
LIN {X -106.6563,Y -87.2776,Z 172,A -138.125,B 8.7929,C 0.3307,E1 8.6764,E2 229.5988} C_DIS
LIN {X -103.7917,Y -90.6655,Z 172,A -136.0793,B 8.7929,C 0.3312,E1 8.6802,E2 227.5281} C_DIS
LIN {X -101.2272,Y -93.5207,Z 172,A -134.583,B 8.7927,C 0.3362,E1 8.683,E2 226.0452} C_DIS
LIN {X -98.0591,Y -96.8376,Z 172,A -132.6337,B 8.7925,C 0.3393,E1 8.6868,E2 224.0911} C_DIS
LIN {X -94.7415,Y -100.0851,Z 172,A -130.7107,B 8.7924,C 0.3431,E1 8.6906,E2 222.1697} C_DIS
LIN {X -91.4548,Y -103.0971,Z 172,A -128.8233,B 8.7923,C 0.346,E1 8.6946,E2 220.2783} C_DIS
LIN {X -87.9151,Y -106.1314,Z 172,A -126.9219,B 8.7921,C 0.3501,E1 8.6986,E2 218.3821} C_DIS
LIN {X -84.538,Y -108.8407,Z 172,A -124.934,B 8.7921,C 0.3498,E1 8.703,E2 216.3705} C_DIS
LIN {X -81.2503,Y -111.3172,Z 172,A -123.3554,B 8.7919,C 0.355,E1 8.7065,E2 214.8093} C_DIS
LIN {X -77.9176,Y -113.674,Z 172,A -121.639,B 8.7919,C 0.3573,E1 8.7105,E2 213.0906} C_DIS
Enddeposition()
END
